  MoveL 7324 to (229.28, 36.09, 106.87) mm, rotated rx -180 ry 0 rz -180 deg; joints [-156.206, -68.965, -50.791, 41.618, 37.406, -35.211]
  MoveL 7325 to (229.28, 36.09, 106.87) mm, rotated rx -180 ry 0 rz -180 deg; joints [-156.206, -68.965, -50.791, 41.618, 37.406, -35.211]
  Call Extruder(199.41394)
  MoveL 7326 to (229.48, 36.14, 106.87) mm, rotated rx -180 ry 0 rz 180 deg; joints [-156.21, -68.992, -50.735, 41.638, 37.382, -35.238]
  MoveL 7327 to (229.48, 36.14, 106.87) mm, rotated rx -180 ry 0 rz 180 deg; joints [-156.21, -68.992, -50.735, 41.638, 37.382, -35.238]
  Call Extruder(199.52925)
  MoveL 7328 to (229.69, 36.18, 106.87) mm, rotated rx 180 ry 0 rz -180 deg; joints [-156.214, -69.019, -50.679, 41.658, 37.357, -35.266]
  MoveL 7329 to (229.69, 36.18, 106.87) mm, rotated rx 180 ry 0 rz -180 deg; joints [-156.214, -69.019, -50.679, 41.658, 37.357, -35.266]
  Call Extruder(199.65431)
  MoveL 7330 to (229.9, 36.25, 106.87) mm, rotated rx 180 ry 0 rz 180 deg; joints [-156.217, -69.048, -50.617, 41.682, 37.331, -35.299]
  MoveL 7331 to (229.9, 36.25, 106.87) mm, rotated rx 180 ry 0 rz 180 deg; joints [-156.217, -69.048, -50.617, 41.682, 37.331, -35.299]
  Call Extruder(199.77989)
  MoveL 7332 to (230.12, 36.31, 106.87) mm, rotated rx -180 ry 0 rz 180 deg; joints [-156.22, -69.077, -50.556, 41.707, 37.305, -35.331]
  MoveL 7333 to (230.12, 36.31, 106.87) mm, rotated rx -180 ry 0 rz 180 deg; joints [-156.22, -69.077, -50.556, 41.707, 37.305, -35.331]
  Call Extruder(199.90597)
  MoveL 7334 to (230.34, 36.37, 106.87) mm, rotated rx 180 ry 0 rz 180 deg; joints [-156.223, -69.106, -50.494, 41.731, 37.279, -35.364]
  MoveL 7335 to (230.34, 36.37, 106.87) mm, rotated rx 180 ry 0 rz 180 deg; joints [-156.223, -69.106, -50.494, 41.731, 37.279, -35.364]
  Call Extruder(200.01064)
  MoveL 7336 to (230.52, 36.43, 106.87) mm, rotated rx 180 ry 0 rz -180 deg; joints [-156.225, -69.131, -50.443, 41.752, 37.258, -35.391]
  MoveL 7337 to (230.52, 36.43, 106.87) mm, rotated rx 180 ry 0 rz -180 deg; joints [-156.225, -69.131, -50.443, 41.752, 37.258, -35.391]
  Call Extruder(200.11570)
  MoveL 7338 to (230.69, 36.49, 106.87) mm, rotated rx 180 ry 0 rz -180 deg; joints [-156.227, -69.155, -50.392, 41.773, 37.237, -35.419]
  MoveL 7339 to (230.69, 36.49, 106.87) mm, rotated rx 180 ry 0 rz -180 deg; joints [-156.227, -69.155, -50.392, 41.773, 37.237, -35.419]
  Call Extruder(200.22759)
  MoveL 7340 to (230.88, 36.55, 106.87) mm, rotated rx 180 ry 0 rz 180 deg; joints [-156.229, -69.181, -50.337, 41.795, 37.214, -35.448]
  MoveL 7341 to (230.88, 36.55, 106.87) mm, rotated rx 180 ry 0 rz 180 deg; joints [-156.229, -69.181, -50.337, 41.795, 37.214, -35.448]
  Call Extruder(200.33994)
  MoveL 7342 to (231.07, 36.61, 106.87) mm, rotated rx -180 ry 0 rz 180 deg; joints [-156.231, -69.207, -50.283, 41.818, 37.192, -35.477]
  MoveL 7343 to (231.07, 36.61, 106.87) mm, rotated rx -180 ry 0 rz 180 deg; joints [-156.231, -69.207, -50.283, 41.818, 37.192, -35.477]
  Call Extruder(200.45272)
  MoveL 7344 to (231.26, 36.67, 106.87) mm, rotated rx -180 ry 0 rz 180 deg; joints [-156.233, -69.232, -50.228, 41.84, 37.17, -35.507]
  MoveL 7345 to (231.26, 36.67, 106.87) mm, rotated rx -180 ry 0 rz 180 deg; joints [-156.233, -69.232, -50.228, 41.84, 37.17, -35.507]
  Call Extruder(200.56596)
  MoveL 7346 to (231.45, 36.73, 106.87) mm, rotated rx 180 ry 0 rz 180 deg; joints [-156.235, -69.258, -50.174, 41.863, 37.147, -35.536]
  MoveL 7347 to (231.45, 36.73, 106.87) mm, rotated rx 180 ry 0 rz 180 deg; joints [-156.235, -69.258, -50.174, 41.863, 37.147, -35.536]
  Call Extruder(200.67963)
  MoveL 7348 to (231.64, 36.79, 106.87) mm, rotated rx 180 ry 0 rz 180 deg; joints [-156.237, -69.284, -50.119, 41.885, 37.125, -35.566]
  MoveL 7349 to (231.64, 36.79, 106.87) mm, rotated rx 180 ry 0 rz 180 deg; joints [-156.237, -69.284, -50.119, 41.885, 37.125, -35.566]
  Call Extruder(200.86159)
  MoveL 7350 to (231.93, 36.91, 106.87) mm, rotated rx 180 ry 0 rz 180 deg; joints [-156.238, -69.326, -50.032, 41.925, 37.09, -35.616]
  MoveL 7351 to (231.93, 36.91, 106.87) mm, rotated rx 180 ry 0 rz 180 deg; joints [-156.238, -69.326, -50.032, 41.925, 37.09, -35.616]
  Call Extruder(201.04431)
  MoveL 7352 to (232.22, 37.03, 106.87) mm, rotated rx 180 ry 0 rz 180 deg; joints [-156.238, -69.367, -49.944, 41.965, 37.055, -35.666]
  MoveL 7353 to (232.22, 37.03, 106.87) mm, rotated rx 180 ry 0 rz 180 deg; joints [-156.238, -69.367, -49.944, 41.965, 37.055, -35.666]
  Call Extruder(201.21473)
  MoveL 7354 to (232.49, 37.15, 106.87) mm, rotated rx 180 ry 0 rz 180 deg; joints [-156.239, -69.406, -49.863, 42.002, 37.023, -35.713]
  MoveL 7355 to (232.49, 37.15, 106.87) mm, rotated rx 180 ry 0 rz 180 deg; joints [-156.239, -69.406, -49.863, 42.002, 37.023, -35.713]
  Call Extruder(201.37273)
  MoveL 7356 to (232.74, 37.26, 106.87) mm, rotated rx 180 ry 0 rz 180 deg; joints [-156.239, -69.442, -49.787, 42.037, 36.994, -35.757]
  MoveL 7357 to (232.74, 37.26, 106.87) mm, rotated rx 180 ry 0 rz 180 deg; joints [-156.239, -69.442, -49.787, 42.037, 36.994, -35.757]
  Call Extruder(201.53133)
  MoveL 7358 to (232.99, 37.36, 106.87) mm, rotated rx -180 ry 0 rz -180 deg; joints [-156.239, -69.478, -49.711, 42.072, 36.964, -35.801]
  MoveL 7359 to (232.99, 37.36, 106.87) mm, rotated rx -180 ry 0 rz -180 deg; joints [-156.239, -69.478, -49.711, 42.072, 36.964, -35.801]
  Call Extruder(201.73750)
  MoveL 7360 to (233.29, 37.54, 106.87) mm, rotated rx 180 ry 0 rz 180 deg; joints [-156.236, -69.524, -49.614, 42.122, 36.928, -35.862]
  MoveL 7361 to (233.29, 37.54, 106.87) mm, rotated rx 180 ry 0 rz 180 deg; joints [-156.236, -69.524, -49.614, 42.122, 36.928, -35.862]
  Call Extruder(201.94444)
  MoveL 7362 to (233.6, 37.71, 106.87) mm, rotated rx -180 ry 0 rz 180 deg; joints [-156.232, -69.57, -49.517, 42.173, 36.893, -35.923]
  MoveL 7363 to (233.6, 37.71, 106.87) mm, rotated rx -180 ry 0 rz 180 deg; joints [-156.232, -69.57, -49.517, 42.173, 36.893, -35.923]
  Call Extruder(202.15217)
  MoveL 7364 to (233.9, 37.89, 106.87) mm, rotated rx -180 ry 0 rz -180 deg; joints [-156.228, -69.617, -49.419, 42.224, 36.857, -35.984]
  MoveL 7365 to (233.9, 37.89, 106.87) mm, rotated rx -180 ry 0 rz -180 deg; joints [-156.228, -69.617, -49.419, 42.224, 36.857, -35.984]
  Call Extruder(202.36067)
  MoveL 7366 to (234.21, 38.06, 106.87) mm, rotated rx 180 ry 0 rz 180 deg; joints [-156.224, -69.663, -49.322, 42.275, 36.821, -36.046]
  MoveL 7367 to (234.21, 38.06, 106.87) mm, rotated rx 180 ry 0 rz 180 deg; joints [-156.224, -69.663, -49.322, 42.275, 36.821, -36.046]
  Call Extruder(202.54021)
  MoveL 7368 to (234.45, 38.24, 106.87) mm, rotated rx -180 ry 0 rz 180 deg; joints [-156.218, -69.703, -49.239, 42.322, 36.793, -36.101]
  MoveL 7369 to (234.45, 38.24, 106.87) mm, rotated rx -180 ry 0 rz 180 deg; joints [-156.218, -69.703, -49.239, 42.322, 36.793, -36.101]
  Call Extruder(202.87363)
  MoveL 7370 to (234.9, 38.57, 106.87) mm, rotated rx 180 ry 0 rz -180 deg; joints [-156.206, -69.776, -49.086, 42.411, 36.741, -36.204]
  MoveL 7371 to (234.9, 38.57, 106.87) mm, rotated rx 180 ry 0 rz -180 deg; joints [-156.206, -69.776, -49.086, 42.411, 36.741, -36.204]
  Call Extruder(203.20823)
  MoveL 7372 to (235.35, 38.9, 106.87) mm, rotated rx -180 ry 0 rz 180 deg; joints [-156.195, -69.849, -48.932, 42.499, 36.688, -36.308]
  Call Extruder(204.03618)
  MoveL 7373 to (236.39, 39.81, 106.87) mm, rotated rx 180 ry 0 rz 180 deg; joints [-156.154, -70.026, -48.56, 42.732, 36.569, -36.573]
  Call Extruder(204.86412)
  MoveL 7374 to (237.3, 40.85, 106.87) mm, rotated rx 180 ry 0 rz 180 deg; joints [-156.097, -70.196, -48.204, 42.98, 36.467, -36.848]
  Call Extruder(205.03142)
  MoveL 7375 to (237.47, 41.07, 106.87) mm, rotated rx 180 ry 0 rz 180 deg; joints [-156.083, -70.229, -48.135, 43.032, 36.449, -36.904]
  MoveL 7376 to (237.47, 41.07, 106.87) mm, rotated rx 180 ry 0 rz 180 deg; joints [-156.083, -70.229, -48.135, 43.032, 36.449, -36.904]
  Call Extruder(205.36483)
  MoveL 7377 to (237.8, 41.52, 106.87) mm, rotated rx 180 ry 0 rz 180 deg; joints [-156.055, -70.295, -47.997, 43.135, 36.412, -37.017]
  MoveL 7378 to (237.8, 41.52, 106.87) mm, rotated rx 180 ry 0 rz 180 deg; joints [-156.055, -70.295, -47.997, 43.135, 36.412, -37.017]
  Call Extruder(205.69706)
  MoveL 7379 to (238.12, 41.98, 106.87) mm, rotated rx 180 ry 0 rz -180 deg; joints [-156.028, -70.361, -47.858, 43.239, 36.376, -37.13]
  MoveL 7380 to (238.12, 41.98, 106.87) mm, rotated rx 180 ry 0 rz -180 deg; joints [-156.028, -70.361, -47.858, 43.239, 36.376, -37.13]
  Call Extruder(205.81476)
  MoveL 7381 to (238.22, 42.15, 106.87) mm, rotated rx -180 ry 0 rz -180 deg; joints [-156.016, -70.383, -47.813, 43.277, 36.366, -37.17]
  MoveL 7382 to (238.22, 42.15, 106.87) mm, rotated rx -180 ry 0 rz -180 deg; joints [-156.016, -70.383, -47.813, 43.277, 36.366, -37.17]
  Call Extruder(206.02249)
  MoveL 7383 to (238.4, 42.45, 106.87) mm, rotated rx 180 ry 0 rz 180 deg; joints [-155.996, -70.422, -47.731, 43.344, 36.347, -37.241]
  MoveL 7384 to (238.4, 42.45, 106.87) mm, rotated rx 180 ry 0 rz 180 deg; joints [-155.996, -70.422, -47.731, 43.344, 36.347, -37.241]
  Call Extruder(206.22943)
  MoveL 7385 to (238.57, 42.75, 106.87) mm, rotated rx -180 ry 0 rz -180 deg; joints [-155.976, -70.461, -47.65, 43.411, 36.328, -37.313]
  MoveL 7386 to (238.57, 42.75, 106.87) mm, rotated rx -180 ry 0 rz -180 deg; joints [-155.976, -70.461, -47.65, 43.411, 36.328, -37.313]
  Call Extruder(206.43560)
  MoveL 7387 to (238.75, 43.06, 106.87) mm, rotated rx 180 ry 0 rz 180 deg; joints [-155.956, -70.5, -47.568, 43.478, 36.31, -37.384]
  MoveL 7388 to (238.75, 43.06, 106.87) mm, rotated rx 180 ry 0 rz 180 deg; joints [-155.956, -70.5, -47.568, 43.478, 36.31, -37.384]
  Call Extruder(206.61728)
  MoveL 7389 to (238.89, 43.33, 106.87) mm, rotated rx 180 ry 0 rz 180 deg; joints [-155.937, -70.533, -47.498, 43.538, 36.295, -37.447]
  MoveL 7390 to (238.89, 43.33, 106.87) mm, rotated rx 180 ry 0 rz 180 deg; joints [-155.937, -70.533, -47.498, 43.538, 36.295, -37.447]
  Call Extruder(206.77529)
  MoveL 7391 to (239, 43.58, 106.87) mm, rotated rx -180 ry 0 rz -180 deg; joints [-155.919, -70.56, -47.441, 43.59, 36.284, -37.501]
  MoveL 7392 to (239, 43.58, 106.87) mm, rotated rx -180 ry 0 rz -180 deg; joints [-155.919, -70.56, -47.441, 43.59, 36.284, -37.501]
  Call Extruder(206.93270)
  MoveL 7393 to (239.1, 43.83, 106.87) mm, rotated rx 180 ry 0 rz -180 deg; joints [-155.901, -70.588, -47.383, 43.642, 36.273, -37.556]
  MoveL 7394 to (239.1, 43.83, 106.87) mm, rotated rx 180 ry 0 rz -180 deg; joints [-155.901, -70.588, -47.383, 43.642, 36.273, -37.556]
  Call Extruder(207.11542)
  MoveL 7395 to (239.23, 44.12, 106.87) mm, rotated rx 180 ry 0 rz 180 deg; joints [-155.879, -70.619, -47.317, 43.703, 36.261, -37.619]
  MoveL 7396 to (239.23, 44.12, 106.87) mm, rotated rx 180 ry 0 rz 180 deg; joints [-155.879, -70.619, -47.317, 43.703, 36.261, -37.619]
  Call Extruder(207.29737)
  MoveL 7397 to (239.35, 44.42, 106.87) mm, rotated rx 180 ry 0 rz -180 deg; joints [-155.858, -70.651, -47.251, 43.764, 36.249, -37.682]
  MoveL 7398 to (239.35, 44.42, 106.87) mm, rotated rx 180 ry 0 rz -180 deg; joints [-155.858, -70.651, -47.251, 43.764, 36.249, -37.682]
  Call Extruder(207.44470)
  MoveL 7399 to (239.44, 44.66, 106.87) mm, rotated rx -180 ry 0 rz -180 deg; joints [-155.84, -70.676, -47.199, 43.814, 36.241, -37.734]
  MoveL 7400 to (239.44, 44.66, 106.87) mm, rotated rx -180 ry 0 rz -180 deg; joints [-155.84, -70.676, -47.199, 43.814, 36.241, -37.734]
  Call Extruder(207.55794)
  MoveL 7401 to (239.5, 44.85, 106.87) mm, rotated rx -180 ry 0 rz 180 deg; joints [-155.826, -70.695, -47.16, 43.852, 36.235, -37.773]
  MoveL 7402 to (239.5, 44.85, 106.87) mm, rotated rx -180 ry 0 rz 180 deg; joints [-155.826, -70.695, -47.16, 43.852, 36.235, -37.773]
  Call Extruder(207.67073)
  MoveL 7403 to (239.56, 45.03, 106.87) mm, rotated rx -180 ry 0 rz 180 deg; joints [-155.811, -70.713, -47.121, 43.89, 36.229, -37.812]
  MoveL 7404 to (239.56, 45.03, 106.87) mm, rotated rx -180 ry 0 rz 180 deg; joints [-155.811, -70.713, -47.121, 43.89, 36.229, -37.812]
  Call Extruder(207.78308)
  MoveL 7405 to (239.62, 45.22, 106.87) mm, rotated rx 180 ry 0 rz -180 deg; joints [-155.797, -70.732, -47.083, 43.929, 36.224, -37.851]
  MoveL 7406 to (239.62, 45.22, 106.87) mm, rotated rx 180 ry 0 rz -180 deg; joints [-155.797, -70.732, -47.083, 43.929, 36.224, -37.851]
  Call Extruder(207.89498)
  MoveL 7407 to (239.68, 45.41, 106.87) mm, rotated rx -180 ry 0 rz 180 deg; joints [-155.783, -70.75, -47.044, 43.967, 36.218, -37.89]
  MoveL 7408 to (239.68, 45.41, 106.87) mm, rotated rx -180 ry 0 rz 180 deg; joints [-155.783, -70.75, -47.044, 43.967, 36.218, -37.89]
  Call Extruder(208.01638)
  MoveL 7409 to (239.75, 45.62, 106.87) mm, rotated rx 180 ry 0 rz 180 deg; joints [-155.767, -70.77, -47.003, 44.009, 36.212, -37.932]
  MoveL 7410 to (239.75, 45.62, 106.87) mm, rotated rx 180 ry 0 rz 180 deg; joints [-155.767, -70.77, -47.003, 44.009, 36.212, -37.932]
  Call Extruder(208.14717)
  MoveL 7411 to (239.81, 45.84, 106.87) mm, rotated rx 180 ry 0 rz 180 deg; joints [-155.75, -70.791, -46.958, 44.054, 36.206, -37.978]
  MoveL 7412 to (239.81, 45.84, 106.87) mm, rotated rx 180 ry 0 rz 180 deg; joints [-155.75, -70.791, -46.958, 44.054, 36.206, -37.978]
  Call Extruder(208.27740)
  MoveL 7413 to (239.88, 46.06, 106.87) mm, rotated rx 180 ry 0 rz 180 deg; joints [-155.733, -70.813, -46.914, 44.099, 36.2, -38.024]
  MoveL 7414 to (239.88, 46.06, 106.87) mm, rotated rx 180 ry 0 rz 180 deg; joints [-155.733, -70.813, -46.914, 44.099, 36.2, -38.024]
  Call Extruder(208.40706)
  MoveL 7415 to (239.95, 46.29, 106.87) mm, rotated rx -180 ry 0 rz 180 deg; joints [-155.715, -70.834, -46.869, 44.144, 36.194, -38.07]
  MoveL 7416 to (239.95, 46.29, 106.87) mm, rotated rx -180 ry 0 rz 180 deg; joints [-155.715, -70.834, -46.869, 44.144, 36.194, -38.07]
  Call Extruder(208.53615)
  MoveL 7417 to (240.02, 46.51, 106.87) mm, rotated rx 180 ry 0 rz 180 deg; joints [-155.698, -70.855, -46.824, 44.189, 36.188, -38.116]
  MoveL 7418 to (240.02, 46.51, 106.87) mm, rotated rx 180 ry 0 rz 180 deg; joints [-155.698, -70.855, -46.824, 44.189, 36.188, -38.116]
  Call Extruder(208.65121)
  MoveL 7419 to (240.06, 46.72, 106.87) mm, rotated rx -180 ry 0 rz -180 deg; joints [-155.682, -70.873, -46.788, 44.229, 36.184, -38.156]
  MoveL 7420 to (240.06, 46.72, 106.87) mm, rotated rx -180 ry 0 rz -180 deg; joints [-155.682, -70.873, -46.788, 44.229, 36.184, -38.156]
  Call Extruder(208.76581)
  MoveL 7421 to (240.11, 46.92, 106.87) mm, rotated rx 180 ry 0 rz -180 deg; joints [-155.665, -70.89, -46.751, 44.269, 36.181, -38.196]
  MoveL 7422 to (240.11, 46.92, 106.87) mm, rotated rx 180 ry 0 rz -180 deg; joints [-155.665, -70.89, -46.751, 44.269, 36.181, -38.196]
  Call Extruder(208.87996)
  MoveL 7423 to (240.15, 47.12, 106.87) mm, rotated rx 180 ry 0 rz 180 deg; joints [-155.649, -70.908, -46.715, 44.308, 36.177, -38.236]
  MoveL 7424 to (240.15, 47.12, 106.87) mm, rotated rx 180 ry 0 rz 180 deg; joints [-155.649, -70.908, -46.715, 44.308, 36.177, -38.236]
  Call Extruder(208.99365)
  MoveL 7425 to (240.2, 47.33, 106.87) mm, rotated rx 180 ry 0 rz 180 deg; joints [-155.633, -70.925, -46.679, 44.348, 36.174, -38.276]
  MoveL 7426 to (240.2, 47.33, 106.87) mm, rotated rx 180 ry 0 rz 180 deg; joints [-155.633, -70.925, -46.679, 44.348, 36.174, -38.276]
  Call Extruder(209.11906)
  MoveL 7427 to (240.24, 47.55, 106.87) mm, rotated rx 180 ry 0 rz 180 deg; joints [-155.614, -70.944, -46.639, 44.392, 36.17, -38.32]
  MoveL 7428 to (240.24, 47.55, 106.87) mm, rotated rx 180 ry 0 rz 180 deg; joints [-155.614, -70.944, -46.639, 44.392, 36.17, -38.32]
  Call Extruder(209.25604)
  MoveL 7429 to (240.29, 47.8, 106.87) mm, rotated rx -180 ry 0 rz 180 deg; joints [-155.594, -70.965, -46.596, 44.441, 36.167, -38.369]
  MoveL 7430 to (240.29, 47.8, 106.87) mm, rotated rx -180 ry 0 rz 180 deg; joints [-155.594, -70.965, -46.596, 44.441, 36.167, -38.369]
  Call Extruder(209.39241)
  MoveL 7431 to (240.34, 48.05, 106.87) mm, rotated rx 180 ry 0 rz 180 deg; joints [-155.574, -70.986, -46.553, 44.489, 36.163, -38.417]
  MoveL 7432 to (240.34, 48.05, 106.87) mm, rotated rx 180 ry 0 rz 180 deg; joints [-155.574, -70.986, -46.553, 44.489, 36.163, -38.417]
  Call Extruder(209.52817)
  MoveL 7433 to (240.39, 48.3, 106.87) mm, rotated rx 180 ry 0 rz 180 deg; joints [-155.554, -71.006, -46.509, 44.538, 36.159, -38.465]
  MoveL 7434 to (240.39, 48.3, 106.87) mm, rotated rx 180 ry 0 rz 180 deg; joints [-155.554, -71.006, -46.509, 44.538, 36.159, -38.465]
  Call Extruder(209.66331)
  MoveL 7435 to (240.44, 48.55, 106.87) mm, rotated rx -180 ry 0 rz 180 deg; joints [-155.534, -71.027, -46.466, 44.586, 36.156, -38.514]
  MoveL 7436 to (240.44, 48.55, 106.87) mm, rotated rx -180 ry 0 rz 180 deg; joints [-155.534, -71.027, -46.466, 44.586, 36.156, -38.514]
  Call Extruder(209.79785)
  MoveL 7437 to (240.49, 48.8, 106.87) mm, rotated rx -180 ry 0 rz -180 deg; joints [-155.514, -71.048, -46.422, 44.634, 36.152, -38.562]
  MoveL 7438 to (240.49, 48.8, 106.87) mm, rotated rx -180 ry 0 rz -180 deg; joints [-155.514, -71.048, -46.422, 44.634, 36.152, -38.562]
  Call Extruder(209.93178)
  MoveL 7439 to (240.54, 49.05, 106.87) mm, rotated rx 180 ry 0 rz 180 deg; joints [-155.494, -71.069, -46.379, 44.683, 36.149, -38.61]
  MoveL 7440 to (240.54, 49.05, 106.87) mm, rotated rx 180 ry 0 rz 180 deg; joints [-155.494, -71.069, -46.379, 44.683, 36.149, -38.61]
  Call Extruder(210.07964)
  MoveL 7441 to (240.59, 49.33, 106.87) mm, rotated rx 180 ry 0 rz 180 deg; joints [-155.471, -71.091, -46.332, 44.736, 36.146, -38.664]
  MoveL 7442 to (240.59, 49.33, 106.87) mm, rotated rx 180 ry 0 rz 180 deg; joints [-155.471, -71.091, -46.332, 44.736, 36.146, -38.664]
  Call Extruder(210.24139)
  MoveL 7443 to (240.64, 49.63, 106.87) mm, rotated rx 180 ry 0 rz -180 deg; joints [-155.446, -71.115, -46.282, 44.794, 36.143, -38.722]
  MoveL 7444 to (240.64, 49.63, 106.87) mm, rotated rx 180 ry 0 rz -180 deg; joints [-155.446, -71.115, -46.282, 44.794, 36.143, -38.722]
  Call Extruder(210.40241)
  MoveL 7445 to (240.69, 49.94, 106.87) mm, rotated rx 180 ry 0 rz 180 deg; joints [-155.421, -71.139, -46.232, 44.853, 36.14, -38.78]
  MoveL 7446 to (240.69, 49.94, 106.87) mm, rotated rx 180 ry 0 rz 180 deg; joints [-155.421, -71.139, -46.232, 44.853, 36.14, -38.78]
  Call Extruder(210.56270)
  MoveL 7447 to (240.74, 50.24, 106.87) mm, rotated rx 180 ry 0 rz 180 deg; joints [-155.396, -71.164, -46.181, 44.911, 36.137, -38.838]
  MoveL 7448 to (240.74, 50.24, 106.87) mm, rotated rx 180 ry 0 rz 180 deg; joints [-155.396, -71.164, -46.181, 44.911, 36.137, -38.838]
  Call Extruder(210.72226)
  MoveL 7449 to (240.78, 50.55, 106.87) mm, rotated rx 180 ry 0 rz 180 deg; joints [-155.371, -71.188, -46.131, 44.97, 36.134, -38.896]
  MoveL 7450 to (240.78, 50.55, 106.87) mm, rotated rx 180 ry 0 rz 180 deg; joints [-155.371, -71.188, -46.131, 44.97, 36.134, -38.896]
  Call Extruder(210.88109)
  MoveL 7451 to (240.83, 50.86, 106.87) mm, rotated rx 180 ry 0 rz 180 deg; joints [-155.346, -71.212, -46.08, 45.028, 36.131, -38.954]
  MoveL 7452 to (240.83, 50.86, 106.87) mm, rotated rx 180 ry 0 rz 180 deg; joints [-155.346, -71.212, -46.08, 45.028, 36.131, -38.954]
  Call Extruder(211.05976)
  MoveL 7453 to (240.88, 51.2, 106.87) mm, rotated rx -180 ry 0 rz -180 deg; joints [-155.317, -71.238, -46.025, 45.094, 36.129, -39.019]
  MoveL 7454 to (240.88, 51.2, 106.87) mm, rotated rx -180 ry 0 rz -180 deg; joints [-155.317, -71.238, -46.025, 45.094, 36.129, -39.019]
  Call Extruder(211.25821)
  MoveL 7455 to (240.93, 51.59, 106.87) mm, rotated rx 180 ry 0 rz -180 deg; joints [-155.285, -71.267, -45.965, 45.167, 36.127, -39.091]
  MoveL 7456 to (240.93, 51.59, 106.87) mm, rotated rx 180 ry 0 rz -180 deg; joints [-155.285, -71.267, -45.965, 45.167, 36.127, -39.091]
  Call Extruder(211.45578)
  MoveL 7457 to (240.97, 51.98, 106.87) mm, rotated rx -180 ry 0 rz 180 deg; joints [-155.252, -71.296, -45.905, 45.24, 36.126, -39.163]
  MoveL 7458 to (240.97, 51.98, 106.87) mm, rotated rx -180 ry 0 rz 180 deg; joints [-155.252, -71.296, -45.905, 45.24, 36.126, -39.163]
  Call Extruder(211.65249)
  MoveL 7459 to (241.02, 52.36, 106.87) mm, rotated rx -180 ry 0 rz 180 deg; joints [-155.22, -71.325, -45.845, 45.313, 36.124, -39.235]
  MoveL 7460 to (241.02, 52.36, 106.87) mm, rotated rx -180 ry 0 rz 180 deg; joints [-155.22, -71.325, -45.845, 45.313, 36.124, -39.235]
  Call Extruder(211.84833)
  MoveL 7461 to (241.06, 52.75, 106.87) mm, rotated rx 180 ry 0 rz 180 deg; joints [-155.188, -71.354, -45.785, 45.386, 36.123, -39.307]
  MoveL 7462 to (241.06, 52.75, 106.87) mm, rotated rx 180 ry 0 rz 180 deg; joints [-155.188, -71.354, -45.785, 45.386, 36.123, -39.307]
  Call Extruder(212.14376)
  MoveL 7463 to (241.11, 53.34, 106.87) mm, rotated rx 180 ry 0 rz 180 deg; joints [-155.138, -71.395, -45.699, 45.495, 36.123, -39.414]
  MoveL 7464 to (241.11, 53.34, 106.87) mm, rotated rx 180 ry 0 rz 180 deg; joints [-155.138, -71.395, -45.699, 45.495, 36.123, -39.414]
  Call Extruder(212.43787)
  MoveL 7465 to (241.16, 53.93, 106.87) mm, rotated rx 180 ry 0 rz 180 deg; joints [-155.088, -71.436, -45.613, 45.604, 36.124, -39.521]
  MoveL 7466 to (241.16, 53.93, 106.87) mm, rotated rx 180 ry 0 rz 180 deg; joints [-155.088, -71.436, -45.613, 45.604, 36.124, -39.521]
  Call Extruder(212.73064)
  MoveL 7467 to (241.2, 54.52, 106.87) mm, rotated rx -180 ry 0 rz -180 deg; joints [-155.038, -71.478, -45.526, 45.713, 36.124, -39.629]
  MoveL 7468 to (241.2, 54.52, 106.87) mm, rotated rx -180 ry 0 rz -180 deg; joints [-155.038, -71.478, -45.526, 45.713, 36.124, -39.629]
  Call Extruder(213.30409)
  MoveL 7469 to (241.25, 55.68, 106.87) mm, rotated rx -180 ry 0 rz -180 deg; joints [-154.938, -71.554, -45.368, 45.925, 36.131, -39.834]
  MoveL 7470 to (241.25, 55.68, 106.87) mm, rotated rx -180 ry 0 rz -180 deg; joints [-154.938, -71.554, -45.368, 45.925, 36.131, -39.834]
  Call Extruder(214.01793)
  MoveL 7471 to (241.29, 57.14, 106.87) mm, rotated rx 180 ry 0 rz 180 deg; joints [-154.812, -71.648, -45.173, 46.188, 36.141, -40.09]
  Call Extruder(256.08281)
  MoveL 7472 to (241.29, 142.86, 106.87) mm, rotated rx 180 ry 0 rz 180 deg; joints [-147.778, -78.434, -31.275, 61.849, 37.21, -56.104]
  Call Extruder(256.51124)
  MoveL 7473 to (241.27, 143.73, 106.87) mm, rotated rx 180 ry 0 rz 180 deg; joints [-147.711, -78.521, -31.1, 62.014, 37.224, -56.283]
  MoveL 7474 to (241.27, 143.73, 106.87) mm, rotated rx 180 ry 0 rz 180 deg; joints [-147.711, -78.521, -31.1, 62.014, 37.224, -56.283]
  Call Extruder(257.08469)
  MoveL 7475 to (241.22, 144.9, 106.87) mm, rotated rx 180 ry 0 rz 180 deg; joints [-147.62, -78.634, -30.873, 62.231, 37.246, -56.517]
  MoveL 7476 to (241.22, 144.9, 106.87) mm, rotated rx 180 ry 0 rz 180 deg; joints [-147.62, -78.634, -30.873, 62.231, 37.246, -56.517]
  Call Extruder(257.51903)
  MoveL 7477 to (241.18, 145.77, 106.87) mm, rotated rx -180 ry 0 rz 180 deg; joints [-147.551, -78.717, -30.704, 62.393, 37.264, -56.691]
  MoveL 7478 to (241.18, 145.77, 106.87) mm, rotated rx -180 ry 0 rz 180 deg; joints [-147.551, -78.717, -30.704, 62.393, 37.264, -56.691]
  Call Extruder(257.81314)
  MoveL 7479 to (241.13, 146.36, 106.87) mm, rotated rx 180 ry 0 rz -180 deg; joints [-147.504, -78.771, -30.595, 62.499, 37.278, -56.805]
  MoveL 7480 to (241.13, 146.36, 106.87) mm, rotated rx 180 ry 0 rz -180 deg; joints [-147.504, -78.771, -30.595, 62.499, 37.278, -56.805]
  Call Extruder(258.10858)
  MoveL 7481 to (241.09, 146.95, 106.87) mm, rotated rx 180 ry 0 rz 180 deg; joints [-147.457, -78.825, -30.486, 62.606, 37.292, -56.92]
  MoveL 7482 to (241.09, 146.95, 106.87) mm, rotated rx 180 ry 0 rz 180 deg; joints [-147.457, -78.825, -30.486, 62.606, 37.292, -56.92]
  Call Extruder(258.35483)
  MoveL 7483 to (241.04, 147.44, 106.87) mm, rotated rx 180 ry 0 rz 180 deg; joints [-147.417, -78.869, -30.397, 62.693, 37.305, -57.013]
  MoveL 7484 to (241.04, 147.44, 106.87) mm, rotated rx 180 ry 0 rz 180 deg; joints [-147.417, -78.869, -30.397, 62.693, 37.305, -57.013]
  Call Extruder(258.55154)
  MoveL 7485 to (240.99, 147.83, 106.87) mm, rotated rx 180 ry 0 rz -180 deg; joints [-147.386, -78.903, -30.33, 62.761, 37.316, -57.086]
  MoveL 7486 to (240.99, 147.83, 106.87) mm, rotated rx 180 ry 0 rz -180 deg; joints [-147.386, -78.903, -30.33, 62.761, 37.316, -57.086]
  Call Extruder(258.74911)
  MoveL 7487 to (240.95, 148.22, 106.87) mm, rotated rx 180 ry 0 rz 180 deg; joints [-147.354, -78.936, -30.263, 62.829, 37.327, -57.158]
  MoveL 7488 to (240.95, 148.22, 106.87) mm, rotated rx 180 ry 0 rz 180 deg; joints [-147.354, -78.936, -30.263, 62.829, 37.327, -57.158]
  Call Extruder(258.94755)
  MoveL 7489 to (240.9, 148.6, 106.87) mm, rotated rx 180 ry 0 rz -180 deg; joints [-147.322, -78.969, -30.195, 62.897, 37.338, -57.23]
  MoveL 7490 to (240.9, 148.6, 106.87) mm, rotated rx 180 ry 0 rz -180 deg; joints [-147.322, -78.969, -30.195, 62.897, 37.338, -57.23]
  Call Extruder(259.14686)
  MoveL 7491 to (240.86, 148.99, 106.87) mm, rotated rx 180 ry 0 rz 180 deg; joints [-147.291, -79.003, -30.128, 62.965, 37.349, -57.303]
  MoveL 7492 to (240.86, 148.99, 106.87) mm, rotated rx 180 ry 0 rz 180 deg; joints [-147.291, -79.003, -30.128, 62.965, 37.349, -57.303]
  Call Extruder(259.30569)
  MoveL 7493 to (240.81, 149.3, 106.87) mm, rotated rx 180 ry 0 rz 180 deg; joints [-147.265, -79.028, -30.078, 63.017, 37.359, -57.357]
  MoveL 7494 to (240.81, 149.3, 106.87) mm, rotated rx 180 ry 0 rz 180 deg; joints [-147.265, -79.028, -30.078, 63.017, 37.359, -57.357]
  Call Extruder(259.46525)
  MoveL 7495 to (240.76, 149.6, 106.87) mm, rotated rx -180 ry 0 rz 180 deg; joints [-147.24, -79.052, -30.028, 63.068, 37.369, -57.412]
  MoveL 7496 to (240.76, 149.6, 106.87) mm, rotated rx -180 ry 0 rz 180 deg; joints [-147.24, -79.052, -30.028, 63.068, 37.369, -57.412]
  Call Extruder(259.62554)
  MoveL 7497 to (240.71, 149.91, 106.87) mm, rotated rx 180 ry 0 rz -180 deg; joints [-147.214, -79.077, -29.979, 63.12, 37.379, -57.467]
  MoveL 7498 to (240.71, 149.91, 106.87) mm, rotated rx 180 ry 0 rz -180 deg; joints [-147.214, -79.077, -29.979, 63.12, 37.379, -57.467]
  Call Extruder(259.78655)
  MoveL 7499 to (240.66, 150.21, 106.87) mm, rotated rx 180 ry 0 rz 180 deg; joints [-147.189, -79.102, -29.929, 63.172, 37.39, -57.521]
  MoveL 7500 to (240.66, 150.21, 106.87) mm, rotated rx 180 ry 0 rz 180 deg; joints [-147.189, -79.102, -29.929, 63.172, 37.39, -57.521]
  Call Extruder(259.94830)
  MoveL 7501 to (240.61, 150.52, 106.87) mm, rotated rx -180 ry 0 rz -180 deg; joints [-147.163, -79.126, -29.879, 63.224, 37.4, -57.576]
  MoveL 7502 to (240.61, 150.52, 106.87) mm, rotated rx -180 ry 0 rz -180 deg; joints [-147.163, -79.126, -29.879, 63.224, 37.4, -57.576]
  Call Extruder(260.11077)
  MoveL 7503 to (240.56, 150.83, 106.87) mm, rotated rx -180 ry 0 rz -180 deg; joints [-147.138, -79.151, -29.829, 63.276, 37.41, -57.631]
  MoveL 7504 to (240.56, 150.83, 106.87) mm, rotated rx -180 ry 0 rz -180 deg; joints [-147.138, -79.151, -29.829, 63.276, 37.41, -57.631]
  Call Extruder(260.24469)
  MoveL 7505 to (240.52, 151.07, 106.87) mm, rotated rx 180 ry 0 rz 180 deg; joints [-147.117, -79.17, -29.791, 63.317, 37.419, -57.674]
  MoveL 7506 to (240.52, 151.07, 106.87) mm, rotated rx 180 ry 0 rz 180 deg; joints [-147.117, -79.17, -29.791, 63.317, 37.419, -57.674]
  Call Extruder(260.37923)
  MoveL 7507 to (240.47, 151.32, 106.87) mm, rotated rx -180 ry 0 rz 180 deg; joints [-147.095, -79.188, -29.754, 63.357, 37.429, -57.716]
  MoveL 7508 to (240.47, 151.32, 106.87) mm, rotated rx -180 ry 0 rz 180 deg; joints [-147.095, -79.188, -29.754, 63.357, 37.429, -57.716]
  Call Extruder(260.51438)
  MoveL 7509 to (240.42, 151.57, 106.87) mm, rotated rx 180 ry 0 rz 180 deg; joints [-147.074, -79.207, -29.717, 63.398, 37.438, -57.759]
  MoveL 7510 to (240.42, 151.57, 106.87) mm, rotated rx 180 ry 0 rz 180 deg; joints [-147.074, -79.207, -29.717, 63.398, 37.438, -57.759]
  Call Extruder(260.65014)
  MoveL 7511 to (240.37, 151.82, 106.87) mm, rotated rx 180 ry 0 rz -180 deg; joints [-147.053, -79.226, -29.679, 63.439, 37.448, -57.802]
  MoveL 7512 to (240.37, 151.82, 106.87) mm, rotated rx 180 ry 0 rz -180 deg; joints [-147.053, -79.226, -29.679, 63.439, 37.448, -57.802]
  Call Extruder(260.78650)
  MoveL 7513 to (240.32, 152.07, 106.87) mm, rotated rx 180 ry 0 rz 180 deg; joints [-147.032, -79.244, -29.641, 63.479, 37.457, -57.844]
  MoveL 7514 to (240.32, 152.07, 106.87) mm, rotated rx 180 ry 0 rz 180 deg; joints [-147.032, -79.244, -29.641, 63.479, 37.457, -57.844]
  Call Extruder(260.92348)
  MoveL 7515 to (240.27, 152.32, 106.87) mm, rotated rx -180 ry 0 rz 180 deg; joints [-147.011, -79.263, -29.603, 63.52, 37.467, -57.887]
  MoveL 7516 to (240.27, 152.32, 106.87) mm, rotated rx -180 ry 0 rz 180 deg; joints [-147.011, -79.263, -29.603, 63.52, 37.467, -57.887]
  Call Extruder(261.06107)
  MoveL 7517 to (240.22, 152.57, 106.87) mm, rotated rx -180 ry 0 rz 180 deg; joints [-146.989, -79.282, -29.566, 63.561, 37.476, -57.929]
  MoveL 7518 to (240.22, 152.57, 106.87) mm, rotated rx -180 ry 0 rz 180 deg; joints [-146.989, -79.282, -29.566, 63.561, 37.476, -57.929]
  Call Extruder(261.17477)
  MoveL 7519 to (240.17, 152.77, 106.87) mm, rotated rx 180 ry 0 rz 180 deg; joints [-146.972, -79.297, -29.536, 63.594, 37.484, -57.964]
  MoveL 7520 to (240.17, 152.77, 106.87) mm, rotated rx 180 ry 0 rz 180 deg; joints [-146.972, -79.297, -29.536, 63.594, 37.484, -57.964]
  Call Extruder(261.28892)
  MoveL 7521 to (240.13, 152.98, 106.87) mm, rotated rx -180 ry 0 rz -180 deg; joints [-146.954, -79.312, -29.506, 63.626, 37.493, -57.998]
  MoveL 7522 to (240.13, 152.98, 106.87) mm, rotated rx -180 ry 0 rz -180 deg; joints [-146.954, -79.312, -29.506, 63.626, 37.493, -57.998]
  Call Extruder(261.40352)
  MoveL 7523 to (240.08, 153.18, 106.87) mm, rotated rx -180 ry 0 rz 180 deg; joints [-146.937, -79.326, -29.476, 63.659, 37.501, -58.032]
  MoveL 7524 to (240.08, 153.18, 106.87) mm, rotated rx -180 ry 0 rz 180 deg; joints [-146.937, -79.326, -29.476, 63.659, 37.501, -58.032]
  Call Extruder(261.51858)
  MoveL 7525 to (240.04, 153.39, 106.87) mm, rotated rx 180 ry 0 rz -180 deg; joints [-146.919, -79.341, -29.446, 63.692, 37.509, -58.066]
  MoveL 7526 to (240.04, 153.39, 106.87) mm, rotated rx 180 ry 0 rz -180 deg; joints [-146.919, -79.341, -29.446, 63.692, 37.509, -58.066]
  Call Extruder(261.64080)
  MoveL 7527 to (239.98, 153.6, 106.87) mm, rotated rx 180 ry 0 rz 180 deg; joints [-146.9, -79.355, -29.418, 63.725, 37.519, -58.1]
  MoveL 7528 to (239.98, 153.6, 106.87) mm, rotated rx 180 ry 0 rz 180 deg; joints [-146.9, -79.355, -29.418, 63.725, 37.519, -58.1]
  Call Extruder(261.77046)
  MoveL 7529 to (239.92, 153.82, 106.87) mm, rotated rx 180 ry 0 rz 180 deg; joints [-146.88, -79.369, -29.392, 63.758, 37.53, -58.134]
  MoveL 7530 to (239.92, 153.82, 106.87) mm, rotated rx 180 ry 0 rz 180 deg; joints [-146.88, -79.369, -29.392, 63.758, 37.53, -58.134]
  Call Extruder(261.90069)
  MoveL 7531 to (239.85, 154.05, 106.87) mm, rotated rx -180 ry 0 rz 180 deg; joints [-146.86, -79.382, -29.366, 63.791, 37.541, -58.167]
  MoveL 7532 to (239.85, 154.05, 106.87) mm, rotated rx -180 ry 0 rz 180 deg; joints [-146.86, -79.382, -29.366, 63.791, 37.541, -58.167]
  Call Extruder(262.03148)
  MoveL 7533 to (239.78, 154.27, 106.87) mm, rotated rx 180 ry 0 rz -180 deg; joints [-146.84, -79.395, -29.339, 63.824, 37.553, -58.201]
  MoveL 7534 to (239.78, 154.27, 106.87) mm, rotated rx 180 ry 0 rz -180 deg; joints [-146.84, -79.395, -29.339, 63.824, 37.553, -58.201]
  Call Extruder(262.16284)
  MoveL 7535 to (239.71, 154.49, 106.87) mm, rotated rx 180 ry 0 rz 180 deg; joints [-146.82, -79.408, -29.312, 63.857, 37.564, -58.234]
  MoveL 7536 to (239.71, 154.49, 106.87) mm, rotated rx 180 ry 0 rz 180 deg; joints [-146.82, -79.408, -29.312, 63.857, 37.564, -58.234]
  Call Extruder(262.27474)
  MoveL 7537 to (239.65, 154.68, 106.87) mm, rotated rx 180 ry 0 rz 180 deg; joints [-146.803, -79.419, -29.291, 63.884, 37.574, -58.261]
  MoveL 7538 to (239.65, 154.68, 106.87) mm, rotated rx 180 ry 0 rz 180 deg; joints [-146.803, -79.419, -29.291, 63.884, 37.574, -58.261]
  Call Extruder(262.38708)
  MoveL 7539 to (239.59, 154.87, 106.87) mm, rotated rx -180 ry 0 rz 180 deg; joints [-146.785, -79.429, -29.27, 63.911, 37.584, -58.289]
  MoveL 7540 to (239.59, 154.87, 106.87) mm, rotated rx -180 ry 0 rz 180 deg; joints [-146.785, -79.429, -29.27, 63.911, 37.584, -58.289]
  Call Extruder(262.49987)
  MoveL 7541 to (239.53, 155.06, 106.87) mm, rotated rx 180 ry 0 rz 180 deg; joints [-146.768, -79.439, -29.249, 63.938, 37.594, -58.316]
  MoveL 7542 to (239.53, 155.06, 106.87) mm, rotated rx 180 ry 0 rz 180 deg; joints [-146.768, -79.439, -29.249, 63.938, 37.594, -58.316]
  Call Extruder(262.61311)
  MoveL 7543 to (239.47, 155.25, 106.87) mm, rotated rx 180 ry 0 rz 180 deg; joints [-146.751, -79.45, -29.228, 63.966, 37.604, -58.343]
  MoveL 7544 to (239.47, 155.25, 106.87) mm, rotated rx 180 ry 0 rz 180 deg; joints [-146.751, -79.45, -29.228, 63.966, 37.604, -58.343]
  Call Extruder(262.72679)
  MoveL 7545 to (239.41, 155.44, 106.87) mm, rotated rx -180 ry 0 rz 180 deg; joints [-146.734, -79.461, -29.207, 63.993, 37.613, -58.371]
  MoveL 7546 to (239.41, 155.44, 106.87) mm, rotated rx -180 ry 0 rz 180 deg; joints [-146.734, -79.461, -29.207, 63.993, 37.613, -58.371]
  Call Extruder(262.90875)
  MoveL 7547 to (239.29, 155.73, 106.87) mm, rotated rx -180 ry 0 rz 180 deg; joints [-146.706, -79.472, -29.183, 64.031, 37.632, -58.407]
  MoveL 7548 to (239.29, 155.73, 106.87) mm, rotated rx -180 ry 0 rz 180 deg; joints [-146.706, -79.472, -29.183, 64.031, 37.632, -58.407]
  Call Extruder(263.09146)
  MoveL 7549 to (239.16, 156.02, 106.87) mm, rotated rx -180 ry 0 rz 180 deg; joints [-146.678, -79.484, -29.159, 64.069, 37.65, -58.444]
  MoveL 7550 to (239.16, 156.02, 106.87) mm, rotated rx -180 ry 0 rz 180 deg; joints [-146.678, -79.484, -29.159, 64.069, 37.65, -58.444]
  Call Extruder(263.26189)
  MoveL 7551 to (239.05, 156.29, 106.87) mm, rotated rx 180 ry 0 rz -180 deg; joints [-146.652, -79.495, -29.137, 64.103, 37.668, -58.478]
  MoveL 7552 to (239.05, 156.29, 106.87) mm, rotated rx 180 ry 0 rz -180 deg; joints [-146.652, -79.495, -29.137, 64.103, 37.668, -58.478]
  Call Extruder(263.41990)
  MoveL 7553 to (238.94, 156.54, 106.87) mm, rotated rx 180 ry 0 rz 180 deg; joints [-146.628, -79.505, -29.118, 64.135, 37.684, -58.508]
  MoveL 7554 to (238.94, 156.54, 106.87) mm, rotated rx 180 ry 0 rz 180 deg; joints [-146.628, -79.505, -29.118, 64.135, 37.684, -58.508]
  Call Extruder(263.57851)
  MoveL 7555 to (238.84, 156.79, 106.87) mm, rotated rx 180 ry 0 rz 180 deg; joints [-146.604, -79.514, -29.098, 64.167, 37.7, -58.539]
  MoveL 7556 to (238.84, 156.79, 106.87) mm, rotated rx 180 ry 0 rz 180 deg; joints [-146.604, -79.514, -29.098, 64.167, 37.7, -58.539]
  Call Extruder(263.78468)
  MoveL 7557 to (238.66, 157.09, 106.87) mm, rotated rx -180 ry 0 rz 180 deg; joints [-146.573, -79.519, -29.09, 64.199, 37.725, -58.566]
  MoveL 7558 to (238.66, 157.09, 106.87) mm, rotated rx -180 ry 0 rz 180 deg; joints [-146.573, -79.519, -29.09, 64.199, 37.725, -58.566]
  Call Extruder(263.99163)
  MoveL 7559 to (238.49, 157.4, 106.87) mm, rotated rx -180 ry 0 rz 180 deg; joints [-146.542, -79.523, -29.081, 64.231, 37.75, -58.594]
  MoveL 7560 to (238.49, 157.4, 106.87) mm, rotated rx -180 ry 0 rz 180 deg; joints [-146.542, -79.523, -29.081, 64.231, 37.75, -58.594]
  Call Extruder(264.19935)
  MoveL 7561 to (238.31, 157.7, 106.87) mm, rotated rx 180 ry 0 rz -180 deg; joints [-146.51, -79.527, -29.072, 64.263, 37.775, -58.621]
  MoveL 7562 to (238.31, 157.7, 106.87) mm, rotated rx 180 ry 0 rz -180 deg; joints [-146.51, -79.527, -29.072, 64.263, 37.775, -58.621]
  Call Extruder(264.40786)
  MoveL 7563 to (238.13, 158.01, 106.87) mm, rotated rx -180 ry 0 rz 180 deg; joints [-146.479, -79.532, -29.064, 64.294, 37.8, -58.649]
  MoveL 7564 to (238.13, 158.01, 106.87) mm, rotated rx -180 ry 0 rz 180 deg; joints [-146.479, -79.532, -29.064, 64.294, 37.8, -58.649]
  Call Extruder(264.58740)
  MoveL 7565 to (237.96, 158.25, 106.87) mm, rotated rx 180 ry 0 rz 180 deg; joints [-146.452, -79.529, -29.068, 64.314, 37.824, -58.664]
  MoveL 7566 to (237.96, 158.25, 106.87) mm, rotated rx 180 ry 0 rz 180 deg; joints [-146.452, -79.529, -29.068, 64.314, 37.824, -58.664]
  Call Extruder(264.92080)
  MoveL 7567 to (237.63, 158.7, 106.87) mm, rotated rx 180 ry 0 rz 180 deg; joints [-146.402, -79.525, -29.078, 64.351, 37.869, -58.69]
  MoveL 7568 to (237.63, 158.7, 106.87) mm, rotated rx 180 ry 0 rz 180 deg; joints [-146.402, -79.525, -29.078, 64.351, 37.869, -58.69]
  Call Extruder(265.25540)
  MoveL 7569 to (237.3, 159.15, 106.87) mm, rotated rx -180 ry 0 rz 180 deg; joints [-146.352, -79.52, -29.087, 64.388, 37.913, -58.716]
  Call Extruder(266.08335)
  MoveL 7570 to (236.39, 160.19, 106.87) mm, rotated rx 180 ry 0 rz 180 deg; joints [-146.229, -79.483, -29.162, 64.448, 38.034, -58.743]
  Call Extruder(266.91129)
  MoveL 7571 to (235.35, 161.1, 106.87) mm, rotated rx -180 ry 0 rz 180 deg; joints [-146.109, -79.412, -29.305, 64.466, 38.168, -58.717]
  Call Extruder(267.07860)
  MoveL 7572 to (235.13, 161.27, 106.87) mm, rotated rx 180 ry 0 rz 180 deg; joints [-146.086, -79.392, -29.344, 64.463, 38.196, -58.704]
  MoveL 7573 to (235.13, 161.27, 106.87) mm, rotated rx 180 ry 0 rz 180 deg; joints [-146.086, -79.392, -29.344, 64.463, 38.196, -58.704]
  Call Extruder(267.41202)
  MoveL 7574 to (234.68, 161.59, 106.87) mm, rotated rx -180 ry 0 rz 180 deg; joints [-146.039, -79.354, -29.421, 64.458, 38.253, -58.678]
  MoveL 7575 to (234.68, 161.59, 106.87) mm, rotated rx -180 ry 0 rz 180 deg; joints [-146.039, -79.354, -29.421, 64.458, 38.253, -58.678]
  Call Extruder(267.74426)
  MoveL 7576 to (234.23, 161.92, 106.87) mm, rotated rx -180 ry 0 rz 180 deg; joints [-145.992, -79.316, -29.498, 64.454, 38.31, -58.653]
  MoveL 7577 to (234.23, 161.92, 106.87) mm, rotated rx -180 ry 0 rz 180 deg; joints [-145.992, -79.316, -29.498, 64.454, 38.31, -58.653]
  Call Extruder(267.86192)
  MoveL 7578 to (234.05, 162.02, 106.87) mm, rotated rx -180 ry 0 rz -180 deg; joints [-145.976, -79.298, -29.533, 64.447, 38.331, -58.638]
  MoveL 7579 to (234.05, 162.02, 106.87) mm, rotated rx -180 ry 0 rz -180 deg; joints [-145.976, -79.298, -29.533, 64.447, 38.331, -58.638]
  Call Extruder(268.06964)
  MoveL 7580 to (233.75, 162.2, 106.87) mm, rotated rx 180 ry 0 rz 180 deg; joints [-145.947, -79.268, -29.595, 64.436, 38.369, -58.612]
  MoveL 7581 to (233.75, 162.2, 106.87) mm, rotated rx 180 ry 0 rz 180 deg; joints [-145.947, -79.268, -29.595, 64.436, 38.369, -58.612]
  Call Extruder(268.27659)
  MoveL 7582 to (233.45, 162.37, 106.87) mm, rotated rx 180 ry 0 rz 180 deg; joints [-145.919, -79.237, -29.657, 64.424, 38.407, -58.585]
  MoveL 7583 to (233.45, 162.37, 106.87) mm, rotated rx 180 ry 0 rz 180 deg; joints [-145.919, -79.237, -29.657, 64.424, 38.407, -58.585]
  Call Extruder(268.48276)
  MoveL 7584 to (233.14, 162.55, 106.87) mm, rotated rx 180 ry 0 rz 180 deg; joints [-145.891, -79.206, -29.718, 64.413, 38.444, -58.559]
  MoveL 7585 to (233.14, 162.55, 106.87) mm, rotated rx 180 ry 0 rz 180 deg; joints [-145.891, -79.206, -29.718, 64.413, 38.444, -58.559]
  Call Extruder(268.66443)
  MoveL 7586 to (232.86, 162.69, 106.87) mm, rotated rx 180 ry 0 rz -180 deg; joints [-145.866, -79.177, -29.778, 64.399, 38.478, -58.531]
  MoveL 7587 to (232.86, 162.69, 106.87) mm, rotated rx 180 ry 0 rz -180 deg; joints [-145.866, -79.177, -29.778, 64.399, 38.478, -58.531]
  Call Extruder(268.82240)
  MoveL 7588 to (232.62, 162.8, 106.87) mm, rotated rx 180 ry 0 rz 180 deg; joints [-145.845, -79.148, -29.837, 64.383, 38.508, -58.502]
  MoveL 7589 to (232.62, 162.8, 106.87) mm, rotated rx 180 ry 0 rz 180 deg; joints [-145.845, -79.148, -29.837, 64.383, 38.508, -58.502]
  Call Extruder(268.97977)
  MoveL 7590 to (232.37, 162.9, 106.87) mm, rotated rx 180 ry 0 rz 180 deg; joints [-145.825, -79.119, -29.895, 64.367, 38.539, -58.473]
  MoveL 7591 to (232.37, 162.9, 106.87) mm, rotated rx 180 ry 0 rz 180 deg; joints [-145.825, -79.119, -29.895, 64.367, 38.539, -58.473]
  Call Extruder(269.16252)
  MoveL 7592 to (232.08, 163.03, 106.87) mm, rotated rx 180 ry 0 rz 180 deg; joints [-145.801, -79.084, -29.964, 64.347, 38.574, -58.438]
  MoveL 7593 to (232.08, 163.03, 106.87) mm, rotated rx 180 ry 0 rz 180 deg; joints [-145.801, -79.084, -29.964, 64.347, 38.574, -58.438]
  Call Extruder(269.34450)
  MoveL 7594 to (231.78, 163.15, 106.87) mm, rotated rx -180 ry 0 rz 180 deg; joints [-145.777, -79.05, -30.033, 64.328, 38.609, -58.403]
  MoveL 7595 to (231.78, 163.15, 106.87) mm, rotated rx -180 ry 0 rz 180 deg; joints [-145.777, -79.05, -30.033, 64.328, 38.609, -58.403]
  Call Extruder(269.49184)
  MoveL 7596 to (231.54, 163.24, 106.87) mm, rotated rx 180 ry 0 rz 180 deg; joints [-145.759, -79.021, -30.092, 64.31, 38.638, -58.373]
  MoveL 7597 to (231.54, 163.24, 106.87) mm, rotated rx 180 ry 0 rz 180 deg; joints [-145.759, -79.021, -30.092, 64.31, 38.638, -58.373]
  Call Extruder(269.60506)
  MoveL 7598 to (231.35, 163.3, 106.87) mm, rotated rx -180 ry 0 rz 180 deg; joints [-145.744, -78.997, -30.14, 64.295, 38.661, -58.347]
  MoveL 7599 to (231.35, 163.3, 106.87) mm, rotated rx -180 ry 0 rz 180 deg; joints [-145.744, -78.997, -30.14, 64.295, 38.661, -58.347]
  Call Extruder(269.71784)
  MoveL 7600 to (231.17, 163.36, 106.87) mm, rotated rx 180 ry 0 rz 180 deg; joints [-145.73, -78.973, -30.188, 64.279, 38.683, -58.322]
  MoveL 7601 to (231.17, 163.36, 106.87) mm, rotated rx 180 ry 0 rz 180 deg; joints [-145.73, -78.973, -30.188, 64.279, 38.683, -58.322]
  Call Extruder(269.83017)
  MoveL 7602 to (230.98, 163.42, 106.87) mm, rotated rx 180 ry 0 rz 180 deg; joints [-145.716, -78.949, -30.237, 64.264, 38.706, -58.296]
  MoveL 7603 to (230.98, 163.42, 106.87) mm, rotated rx 180 ry 0 rz 180 deg; joints [-145.716, -78.949, -30.237, 64.264, 38.706, -58.296]
  Call Extruder(269.94206)
  MoveL 7604 to (230.79, 163.48, 106.87) mm, rotated rx 180 ry 0 rz 180 deg; joints [-145.702, -78.925, -30.284, 64.249, 38.728, -58.27]
  MoveL 7605 to (230.79, 163.48, 106.87) mm, rotated rx 180 ry 0 rz 180 deg; joints [-145.702, -78.925, -30.284, 64.249, 38.728, -58.27]
  Call Extruder(270.06346)
  MoveL 7606 to (230.58, 163.55, 106.87) mm, rotated rx -180 ry 0 rz 180 deg; joints [-145.687, -78.899, -30.337, 64.232, 38.753, -58.242]
  MoveL 7607 to (230.58, 163.55, 106.87) mm, rotated rx -180 ry 0 rz 180 deg; joints [-145.687, -78.899, -30.337, 64.232, 38.753, -58.242]
  Call Extruder(270.19428)
  MoveL 7608 to (230.36, 163.61, 106.87) mm, rotated rx 180 ry 0 rz -180 deg; joints [-145.67, -78.87, -30.395, 64.213, 38.78, -58.211]
  MoveL 7609 to (230.36, 163.61, 106.87) mm, rotated rx 180 ry 0 rz -180 deg; joints [-145.67, -78.87, -30.395, 64.213, 38.78, -58.211]
  Call Extruder(270.32452)
  MoveL 7610 to (230.14, 163.68, 106.87) mm, rotated rx -180 ry 0 rz 180 deg; joints [-145.654, -78.842, -30.453, 64.194, 38.806, -58.18]
  MoveL 7611 to (230.14, 163.68, 106.87) mm, rotated rx -180 ry 0 rz 180 deg; joints [-145.654, -78.842, -30.453, 64.194, 38.806, -58.18]
  Call Extruder(270.45421)
  MoveL 7612 to (229.91, 163.75, 106.87) mm, rotated rx 180 ry 0 rz 180 deg; joints [-145.638, -78.813, -30.511, 64.175, 38.833, -58.149]
  MoveL 7613 to (229.91, 163.75, 106.87) mm, rotated rx 180 ry 0 rz 180 deg; joints [-145.638, -78.813, -30.511, 64.175, 38.833, -58.149]
  Call Extruder(270.58333)
  MoveL 7614 to (229.69, 163.82, 106.87) mm, rotated rx -180 ry 0 rz 180 deg; joints [-145.621, -78.784, -30.569, 64.156, 38.859, -58.118]
  MoveL 7615 to (229.69, 163.82, 106.87) mm, rotated rx -180 ry 0 rz 180 deg; joints [-145.621, -78.784, -30.569, 64.156, 38.859, -58.118]
  Call Extruder(270.69840)
  MoveL 7616 to (229.48, 163.86, 106.87) mm, rotated rx -180 ry 0 rz 180 deg; joints [-145.607, -78.756, -30.625, 64.136, 38.883, -58.086]
  MoveL 7617 to (229.48, 163.86, 106.87) mm, rotated rx -180 ry 0 rz 180 deg; joints [-145.607, -78.756, -30.625, 64.136, 38.883, -58.086]
  Call Extruder(270.81302)
  MoveL 7618 to (229.28, 163.91, 106.87) mm, rotated rx 180 ry 0 rz -180 deg; joints [-145.594, -78.728, -30.681, 64.116, 38.907, -58.054]
  MoveL 7619 to (229.28, 163.91, 106.87) mm, rotated rx 180 ry 0 rz -180 deg; joints [-145.594, -78.728, -30.681, 64.116, 38.907, -58.054]
  Call Extruder(270.92719)
  MoveL 7620 to (229.08, 163.95, 106.87) mm, rotated rx -180 ry 0 rz 180 deg; joints [-145.58, -78.701, -30.737, 64.096, 38.931, -58.023]
  MoveL 7621 to (229.08, 163.95, 106.87) mm, rotated rx -180 ry 0 rz 180 deg; joints [-145.58, -78.701, -30.737, 64.096, 38.931, -58.023]
  Call Extruder(271.04091)
  MoveL 7622 to (228.87, 164, 106.87) mm, rotated rx 180 ry 0 rz -180 deg; joints [-145.566, -78.673, -30.793, 64.076, 38.956, -57.991]
  MoveL 7623 to (228.87, 164, 106.87) mm, rotated rx 180 ry 0 rz -180 deg; joints [-145.566, -78.673, -30.793, 64.076, 38.956, -57.991]
  Call Extruder(271.16633)
  MoveL 7624 to (228.65, 164.04, 106.87) mm, rotated rx -180 ry 0 rz 180 deg; joints [-145.551, -78.642, -30.856, 64.054, 38.982, -57.956]
  MoveL 7625 to (228.65, 164.04, 106.87) mm, rotated rx -180 ry 0 rz 180 deg; joints [-145.551, -78.642, -30.856, 64.054, 38.982, -57.956]
  Call Extruder(271.30331)
  MoveL 7626 to (228.4, 164.09, 106.87) mm, rotated rx 180 ry 0 rz 180 deg; joints [-145.535, -78.607, -30.925, 64.029, 39.011, -57.917]
  MoveL 7627 to (228.4, 164.09, 106.87) mm, rotated rx 180 ry 0 rz 180 deg; joints [-145.535, -78.607, -30.925, 64.029, 39.011, -57.917]
  Call Extruder(271.43968)
  MoveL 7628 to (228.15, 164.14, 106.87) mm, rotated rx 180 ry 0 rz 180 deg; joints [-145.518, -78.573, -30.995, 64.004, 39.041, -57.878]
  MoveL 7629 to (228.15, 164.14, 106.87) mm, rotated rx 180 ry 0 rz 180 deg; joints [-145.518, -78.573, -30.995, 64.004, 39.041, -57.878]
  Call Extruder(271.57543)
  MoveL 7630 to (227.9, 164.19, 106.87) mm, rotated rx -180 ry 0 rz 180 deg; joints [-145.502, -78.539, -31.064, 63.979, 39.07, -57.839]
  MoveL 7631 to (227.9, 164.19, 106.87) mm, rotated rx -180 ry 0 rz 180 deg; joints [-145.502, -78.539, -31.064, 63.979, 39.07, -57.839]
  Call Extruder(271.71058)
  MoveL 7632 to (227.65, 164.24, 106.87) mm, rotated rx 180 ry 0 rz 180 deg; joints [-145.485, -78.505, -31.133, 63.955, 39.099, -57.8]
  MoveL 7633 to (227.65, 164.24, 106.87) mm, rotated rx 180 ry 0 rz 180 deg; joints [-145.485, -78.505, -31.133, 63.955, 39.099, -57.8]
  Call Extruder(271.84512)
  MoveL 7634 to (227.4, 164.29, 106.87) mm, rotated rx 180 ry 0 rz 180 deg; joints [-145.469, -78.471, -31.201, 63.93, 39.128, -57.762]
  MoveL 7635 to (227.4, 164.29, 106.87) mm, rotated rx 180 ry 0 rz 180 deg; joints [-145.469, -78.471, -31.201, 63.93, 39.128, -57.762]
  Call Extruder(271.97904)
  MoveL 7636 to (227.15, 164.34, 106.87) mm, rotated rx 180 ry 0 rz 180 deg; joints [-145.453, -78.437, -31.27, 63.906, 39.157, -57.723]
  MoveL 7637 to (227.15, 164.34, 106.87) mm, rotated rx 180 ry 0 rz 180 deg; joints [-145.453, -78.437, -31.27, 63.906, 39.157, -57.723]
  Call Extruder(272.12691)
  MoveL 7638 to (226.87, 164.39, 106.87) mm, rotated rx 180 ry 0 rz -180 deg; joints [-145.435, -78.398, -31.347, 63.878, 39.189, -57.679]
  MoveL 7639 to (226.87, 164.39, 106.87) mm, rotated rx 180 ry 0 rz -180 deg; joints [-145.435, -78.398, -31.347, 63.878, 39.189, -57.679]
  Call Extruder(272.28865)
  MoveL 7640 to (226.57, 164.44, 106.87) mm, rotated rx 180 ry 0 rz 180 deg; joints [-145.415, -78.355, -31.434, 63.846, 39.225, -57.63]
  MoveL 7641 to (226.57, 164.44, 106.87) mm, rotated rx 180 ry 0 rz 180 deg; joints [-145.415, -78.355, -31.434, 63.846, 39.225, -57.63]
  Call Extruder(272.44966)
  MoveL 7642 to (226.26, 164.49, 106.87) mm, rotated rx -180 ry 0 rz 180 deg; joints [-145.396, -78.312, -31.521, 63.815, 39.261, -57.58]
  MoveL 7643 to (226.26, 164.49, 106.87) mm, rotated rx -180 ry 0 rz 180 deg; joints [-145.396, -78.312, -31.521, 63.815, 39.261, -57.58]
  Call Extruder(272.60995)
  MoveL 7644 to (225.96, 164.53, 106.87) mm, rotated rx 180 ry 0 rz 180 deg; joints [-145.377, -78.27, -31.607, 63.783, 39.296, -57.531]
  MoveL 7645 to (225.96, 164.53, 106.87) mm, rotated rx 180 ry 0 rz 180 deg; joints [-145.377, -78.27, -31.607, 63.783, 39.296, -57.531]
  Call Extruder(272.76951)
  MoveL 7646 to (225.65, 164.58, 106.87) mm, rotated rx -180 ry 0 rz -180 deg; joints [-145.357, -78.227, -31.693, 63.752, 39.332, -57.483]
  MoveL 7647 to (225.65, 164.58, 106.87) mm, rotated rx -180 ry 0 rz -180 deg; joints [-145.357, -78.227, -31.693, 63.752, 39.332, -57.483]
  Call Extruder(272.92834)
  MoveL 7648 to (225.34, 164.63, 106.87) mm, rotated rx 180 ry 0 rz 180 deg; joints [-145.338, -78.185, -31.779, 63.721, 39.367, -57.434]
  MoveL 7649 to (225.34, 164.63, 106.87) mm, rotated rx 180 ry 0 rz 180 deg; joints [-145.338, -78.185, -31.779, 63.721, 39.367, -57.434]
  Call Extruder(273.10701)
  MoveL 7650 to (225, 164.68, 106.87) mm, rotated rx -180 ry 0 rz 180 deg; joints [-145.317, -78.136, -31.878, 63.685, 39.407, -57.377]
  MoveL 7651 to (225, 164.68, 106.87) mm, rotated rx -180 ry 0 rz 180 deg; joints [-145.317, -78.136, -31.878, 63.685, 39.407, -57.377]
  Call Extruder(273.30545)
  MoveL 7652 to (224.61, 164.72, 106.87) mm, rotated rx -180 ry 0 rz 180 deg; joints [-145.293, -78.081, -31.989, 63.643, 39.452, -57.313]
  MoveL 7653 to (224.61, 164.72, 106.87) mm, rotated rx -180 ry 0 rz 180 deg; joints [-145.293, -78.081, -31.989, 63.643, 39.452, -57.313]
  Call Extruder(273.50302)
  MoveL 7654 to (224.22, 164.77, 106.87) mm, rotated rx -180 ry 0 rz 180 deg; joints [-145.27, -78.026, -32.101, 63.602, 39.497, -57.249]
  MoveL 7655 to (224.22, 164.77, 106.87) mm, rotated rx -180 ry 0 rz 180 deg; joints [-145.27, -78.026, -32.101, 63.602, 39.497, -57.249]
  Call Extruder(273.69973)
  MoveL 7656 to (223.84, 164.82, 106.87) mm, rotated rx 180 ry 0 rz 180 deg; joints [-145.246, -77.971, -32.211, 63.561, 39.542, -57.186]
  MoveL 7657 to (223.84, 164.82, 106.87) mm, rotated rx 180 ry 0 rz 180 deg; joints [-145.246, -77.971, -32.211, 63.561, 39.542, -57.186]
  Call Extruder(273.89557)
  MoveL 7658 to (223.45, 164.86, 106.87) mm, rotated rx 180 ry 0 rz 180 deg; joints [-145.223, -77.916, -32.323, 63.52, 39.586, -57.122]
  MoveL 7659 to (223.45, 164.86, 106.87) mm, rotated rx 180 ry 0 rz 180 deg; joints [-145.223, -77.916, -32.323, 63.52, 39.586, -57.122]
  Call Extruder(274.19092)
  MoveL 7660 to (222.86, 164.91, 106.87) mm, rotated rx -180 ry 0 rz 180 deg; joints [-145.189, -77.83, -32.495, 63.455, 39.654, -57.022]
  MoveL 7661 to (222.86, 164.91, 106.87) mm, rotated rx -180 ry 0 rz 180 deg; joints [-145.189, -77.83, -32.495, 63.455, 39.654, -57.022]
  Call Extruder(274.48494)
  MoveL 7662 to (222.27, 164.96, 106.87) mm, rotated rx 180 ry 0 rz 180 deg; joints [-145.155, -77.745, -32.667, 63.39, 39.721, -56.922]
  MoveL 7663 to (222.27, 164.96, 106.87) mm, rotated rx 180 ry 0 rz 180 deg; joints [-145.155, -77.745, -32.667, 63.39, 39.721, -56.922]
  Call Extruder(274.77764)
  MoveL 7664 to (221.68, 165, 106.87) mm, rotated rx 180 ry 0 rz 180 deg; joints [-145.121, -77.661, -32.839, 63.326, 39.789, -56.824]
  MoveL 7665 to (221.68, 165, 106.87) mm, rotated rx 180 ry 0 rz 180 deg; joints [-145.121, -77.661, -32.839, 63.326, 39.789, -56.824]
  Call Extruder(275.35108)
  MoveL 7666 to (220.52, 165.05, 106.87) mm, rotated rx 180 ry 0 rz 180 deg; joints [-145.056, -77.49, -33.185, 63.193, 39.921, -56.621]
  MoveL 7667 to (220.52, 165.05, 106.87) mm, rotated rx 180 ry 0 rz 180 deg; joints [-145.056, -77.49, -33.185, 63.193, 39.921, -56.621]
  Call Extruder(276.06510)
  MoveL 7668 to (219.06, 165.09, 106.87) mm, rotated rx 180 ry 0 rz 180 deg; joints [-144.977, -77.277, -33.617, 63.028, 40.086, -56.369]
  Call Extruder(392.91185)
  MoveL 7669 to (-19.06, 165.09, 106.87) mm, rotated rx 180 ry 0 rz -180 deg; joints [-127.435, -56.551, -78.268, 61.649, 64.458, -38.627]
  Call Extruder(393.34045)
  MoveL 7670 to (-19.94, 165.07, 106.87) mm, rotated rx -180 ry 0 rz -180 deg; joints [-127.348, -56.505, -78.377, 61.697, 64.542, -38.598]
  MoveL 7671 to (-19.94, 165.07, 106.87) mm, rotated rx -180 ry 0 rz -180 deg; joints [-127.348, -56.505, -78.377, 61.697, 64.542, -38.598]
  Call Extruder(393.91390)
  MoveL 7672 to (-21.1, 165.02, 106.87) mm, rotated rx 180 ry 0 rz 180 deg; joints [-127.235, -56.443, -78.525, 61.76, 64.653, -38.557]
  MoveL 7673 to (-21.1, 165.02, 106.87) mm, rotated rx 180 ry 0 rz 180 deg; joints [-127.235, -56.443, -78.525, 61.76, 64.653, -38.557]
  Call Extruder(394.34820)
  MoveL 7674 to (-21.97, 164.98, 106.87) mm, rotated rx 180 ry 0 rz 180 deg; joints [-127.15, -56.395, -78.638, 61.807, 64.737, -38.525]
  MoveL 7675 to (-21.97, 164.98, 106.87) mm, rotated rx 180 ry 0 rz 180 deg; joints [-127.15, -56.395, -78.638, 61.807, 64.737, -38.525]
  Call Extruder(394.64223)
  MoveL 7676 to (-22.56, 164.93, 106.87) mm, rotated rx 180 ry 0 rz -180 deg; joints [-127.093, -56.362, -78.716, 61.836, 64.793, -38.502]
  MoveL 7677 to (-22.56, 164.93, 106.87) mm, rotated rx 180 ry 0 rz -180 deg; joints [-127.093, -56.362, -78.716, 61.836, 64.793, -38.502]
  Call Extruder(394.93759)
  MoveL 7678 to (-23.15, 164.89, 106.87) mm, rotated rx 180 ry 0 rz 180 deg; joints [-127.037, -56.329, -78.794, 61.866, 64.849, -38.478]
  MoveL 7679 to (-23.15, 164.89, 106.87) mm, rotated rx 180 ry 0 rz 180 deg; joints [-127.037, -56.329, -78.794, 61.866, 64.849, -38.478]
  Call Extruder(395.18380)
  MoveL 7680 to (-23.64, 164.84, 106.87) mm, rotated rx 180 ry 0 rz 180 deg; joints [-126.991, -56.301, -78.86, 61.89, 64.896, -38.458]
  MoveL 7681 to (-23.64, 164.84, 106.87) mm, rotated rx 180 ry 0 rz 180 deg; joints [-126.991, -56.301, -78.86, 61.89, 64.896, -38.458]
  Call Extruder(395.38051)
  MoveL 7682 to (-24.03, 164.79, 106.87) mm, rotated rx 180 ry 0 rz 180 deg; joints [-126.955, -56.279, -78.914, 61.909, 64.933, -38.441]
  MoveL 7683 to (-24.03, 164.79, 106.87) mm, rotated rx 180 ry 0 rz 180 deg; joints [-126.955, -56.279, -78.914, 61.909, 64.933, -38.441]
  Call Extruder(395.57808)
  MoveL 7684 to (-24.42, 164.75, 106.87) mm, rotated rx 180 ry 0 rz -180 deg; joints [-126.919, -56.256, -78.967, 61.927, 64.97, -38.424]
  MoveL 7685 to (-24.42, 164.75, 106.87) mm, rotated rx 180 ry 0 rz -180 deg; joints [-126.919, -56.256, -78.967, 61.927, 64.97, -38.424]
  Call Extruder(395.77652)
  MoveL 7686 to (-24.8, 164.7, 106.87) mm, rotated rx -180 ry 0 rz 180 deg; joints [-126.883, -56.233, -79.021, 61.945, 65.007, -38.407]
  MoveL 7687 to (-24.8, 164.7, 106.87) mm, rotated rx -180 ry 0 rz 180 deg; joints [-126.883, -56.233, -79.021, 61.945, 65.007, -38.407]
  Call Extruder(395.97583)
  MoveL 7688 to (-25.19, 164.66, 106.87) mm, rotated rx -180 ry 0 rz 180 deg; joints [-126.847, -56.211, -79.074, 61.964, 65.044, -38.39]
  MoveL 7689 to (-25.19, 164.66, 106.87) mm, rotated rx -180 ry 0 rz 180 deg; joints [-126.847, -56.211, -79.074, 61.964, 65.044, -38.39]
  Call Extruder(396.13466)
  MoveL 7690 to (-25.5, 164.61, 106.87) mm, rotated rx 180 ry 0 rz 180 deg; joints [-126.82, -56.192, -79.118, 61.977, 65.073, -38.376]
  MoveL 7691 to (-25.5, 164.61, 106.87) mm, rotated rx 180 ry 0 rz 180 deg; joints [-126.82, -56.192, -79.118, 61.977, 65.073, -38.376]
  Call Extruder(396.29423)
  MoveL 7692 to (-25.8, 164.56, 106.87) mm, rotated rx 180 ry 0 rz 180 deg; joints [-126.792, -56.174, -79.162, 61.99, 65.102, -38.361]
  MoveL 7693 to (-25.8, 164.56, 106.87) mm, rotated rx 180 ry 0 rz 180 deg; joints [-126.792, -56.174, -79.162, 61.99, 65.102, -38.361]
  Call Extruder(396.45451)
  MoveL 7694 to (-26.11, 164.51, 106.87) mm, rotated rx -180 ry 0 rz 180 deg; joints [-126.765, -56.155, -79.206, 62.004, 65.131, -38.346]
  MoveL 7695 to (-26.11, 164.51, 106.87) mm, rotated rx -180 ry 0 rz 180 deg; joints [-126.765, -56.155, -79.206, 62.004, 65.131, -38.346]
  Call Extruder(396.61553)
  MoveL 7696 to (-26.41, 164.46, 106.87) mm, rotated rx -180 ry 0 rz 180 deg; joints [-126.737, -56.137, -79.25, 62.017, 65.16, -38.331]
  MoveL 7697 to (-26.41, 164.46, 106.87) mm, rotated rx -180 ry 0 rz 180 deg; joints [-126.737, -56.137, -79.25, 62.017, 65.16, -38.331]
  Call Extruder(396.77727)
  MoveL 7698 to (-26.72, 164.41, 106.87) mm, rotated rx 180 ry 0 rz 180 deg; joints [-126.71, -56.118, -79.294, 62.031, 65.189, -38.317]
  MoveL 7699 to (-26.72, 164.41, 106.87) mm, rotated rx 180 ry 0 rz 180 deg; joints [-126.71, -56.118, -79.294, 62.031, 65.189, -38.317]
  Call Extruder(396.93974)
  MoveL 7700 to (-27.03, 164.37, 106.87) mm, rotated rx 180 ry 0 rz 180 deg; joints [-126.682, -56.1, -79.338, 62.044, 65.218, -38.302]
  MoveL 7701 to (-27.03, 164.37, 106.87) mm, rotated rx 180 ry 0 rz 180 deg; joints [-126.682, -56.1, -79.338, 62.044, 65.218, -38.302]
  Call Extruder(397.07367)
  MoveL 7702 to (-27.27, 164.32, 106.87) mm, rotated rx 180 ry 0 rz 180 deg; joints [-126.66, -56.084, -79.375, 62.054, 65.242, -38.289]
  MoveL 7703 to (-27.27, 164.32, 106.87) mm, rotated rx 180 ry 0 rz 180 deg; joints [-126.66, -56.084, -79.375, 62.054, 65.242, -38.289]
  Call Extruder(397.20821)
  MoveL 7704 to (-27.52, 164.27, 106.87) mm, rotated rx 180 ry 0 rz 180 deg; joints [-126.638, -56.068, -79.413, 62.064, 65.265, -38.275]
  MoveL 7705 to (-27.52, 164.27, 106.87) mm, rotated rx 180 ry 0 rz 180 deg; joints [-126.638, -56.068, -79.413, 62.064, 65.265, -38.275]
  Call Extruder(397.34335)
  MoveL 7706 to (-27.77, 164.22, 106.87) mm, rotated rx -180 ry 0 rz -180 deg; joints [-126.617, -56.053, -79.45, 62.074, 65.289, -38.262]
  MoveL 7707 to (-27.77, 164.22, 106.87) mm, rotated rx -180 ry 0 rz -180 deg; joints [-126.617, -56.053, -79.45, 62.074, 65.289, -38.262]
  Call Extruder(397.47911)
  MoveL 7708 to (-28.02, 164.17, 106.87) mm, rotated rx -180 ry 0 rz 180 deg; joints [-126.595, -56.037, -79.487, 62.084, 65.312, -38.249]
  MoveL 7709 to (-28.02, 164.17, 106.87) mm, rotated rx -180 ry 0 rz 180 deg; joints [-126.595, -56.037, -79.487, 62.084, 65.312, -38.249]
  Call Extruder(397.61548)
  MoveL 7710 to (-28.27, 164.12, 106.87) mm, rotated rx -180 ry 0 rz 180 deg; joints [-126.573, -56.021, -79.524, 62.094, 65.336, -38.236]
  MoveL 7711 to (-28.27, 164.12, 106.87) mm, rotated rx -180 ry 0 rz 180 deg; joints [-126.573, -56.021, -79.524, 62.094, 65.336, -38.236]
  Call Extruder(397.70034)
  MoveL 7712 to (-28.43, 164.09, 106.87) mm, rotated rx 180 ry 0 rz 180 deg; joints [-126.559, -56.012, -79.547, 62.101, 65.351, -38.228]
  Set speed (130.0 mm/s)
  MoveL 7713 to (-31.76, 163.31, 106.87) mm, rotated rx 180 ry 0 rz 180 deg; joints [-126.274, -55.796, -80.061, 62.227, 65.666, -38.041]
  MoveL 7714 to (-31.76, 163.31, 116.27) mm, rotated rx 180 ry 0 rz -180 deg; joints [-126.274, -54.543, -80.572, 62.527, 65.322, -38.764]
  Call Extruder(395.70034)
  Set speed (40.0 mm/s)
  MoveL 7715 to (-31.76, 163.31, 116.27) mm, rotated rx 180 ry 0 rz -180 deg; joints [-126.274, -54.543, -80.572, 62.527, 65.322, -38.764]
  Call Extruder(0.00000)
  Set speed (130.0 mm/s)
  MoveL 7716 to (-34.22, 161.92, 116.27) mm, rotated rx -180 ry 0 rz 180 deg; joints [-126.122, -54.327, -81.077, 62.54, 65.55, -38.535]
  Call Extruder(2.00000)
  Set speed (40.0 mm/s)
  MoveL 7717 to (-34.22, 161.92, 116.27) mm, rotated rx -180 ry 0 rz 180 deg; joints [-126.122, -54.327, -81.077, 62.54, 65.55, -38.535]
  Set speed (30.0 mm/s)
  MoveL 7718 to (-34.22, 161.92, 116.27) mm, rotated rx -180 ry 0 rz 180 deg; joints [-126.122, -54.327, -81.077, 62.54, 65.55, -38.535]
  Call Extruder(2.16612)
  MoveL 7719 to (-34.45, 161.76, 116.27) mm, rotated rx -180 ry 0 rz 180 deg; joints [-126.111, -54.305, -81.13, 62.537, 65.571, -38.51]
  MoveL 7720 to (-34.45, 161.76, 116.27) mm, rotated rx -180 ry 0 rz 180 deg; joints [-126.111, -54.305, -81.13, 62.537, 65.571, -38.51]
  Call Extruder(2.49954)
  MoveL 7721 to (-34.9, 161.43, 116.27) mm, rotated rx -180 ry 0 rz 180 deg; joints [-126.089, -54.26, -81.233, 62.533, 65.612, -38.46]
  MoveL 7722 to (-34.9, 161.43, 116.27) mm, rotated rx -180 ry 0 rz 180 deg; joints [-126.089, -54.26, -81.233, 62.533, 65.612, -38.46]
  Call Extruder(2.83415)
  MoveL 7723 to (-35.35, 161.1, 116.27) mm, rotated rx 180 ry 0 rz 180 deg; joints [-126.067, -54.216, -81.337, 62.528, 65.654, -38.41]
  Call Extruder(3.66207)
  MoveL 7724 to (-36.39, 160.19, 116.27) mm, rotated rx 180 ry 0 rz 180 deg; joints [-126.027, -54.104, -81.6, 62.501, 65.748, -38.277]
  Call Extruder(4.49000)
  MoveL 7725 to (-37.3, 159.15, 116.27) mm, rotated rx 180 ry 0 rz 180 deg; joints [-126.011, -53.99, -81.868, 62.454, 65.829, -38.133]
  Call Extruder(4.65731)
  MoveL 7726 to (-37.47, 158.93, 116.27) mm, rotated rx -180 ry 0 rz 180 deg; joints [-126.011, -53.967, -81.923, 62.442, 65.844, -38.102]
  MoveL 7727 to (-37.47, 158.93, 116.27) mm, rotated rx -180 ry 0 rz 180 deg; joints [-126.011, -53.967, -81.923, 62.442, 65.844, -38.102]
  Call Extruder(4.99074)
  MoveL 7728 to (-37.79, 158.48, 116.27) mm, rotated rx 180 ry 0 rz 180 deg; joints [-126.011, -53.921, -82.031, 62.417, 65.873, -38.041]
  MoveL 7729 to (-37.79, 158.48, 116.27) mm, rotated rx 180 ry 0 rz 180 deg; joints [-126.011, -53.921, -82.031, 62.417, 65.873, -38.041]
  Call Extruder(5.32299)
  MoveL 7730 to (-38.12, 158.02, 116.27) mm, rotated rx -180 ry 0 rz 180 deg; joints [-126.011, -53.876, -82.14, 62.392, 65.902, -37.981]
  MoveL 7731 to (-38.12, 158.02, 116.27) mm, rotated rx -180 ry 0 rz 180 deg; joints [-126.011, -53.876, -82.14, 62.392, 65.902, -37.981]
  Call Extruder(5.44066)
  MoveL 7732 to (-38.22, 157.85, 116.27) mm, rotated rx 180 ry 0 rz 180 deg; joints [-126.013, -53.859, -82.178, 62.381, 65.91, -37.958]
  MoveL 7733 to (-38.22, 157.85, 116.27) mm, rotated rx 180 ry 0 rz 180 deg; joints [-126.013, -53.859, -82.178, 62.381, 65.91, -37.958]
  Call Extruder(5.64838)
  MoveL 7734 to (-38.4, 157.55, 116.27) mm, rotated rx 180 ry 0 rz 180 deg; joints [-126.018, -53.831, -82.245, 62.361, 65.925, -37.919]
  MoveL 7735 to (-38.4, 157.55, 116.27) mm, rotated rx 180 ry 0 rz 180 deg; joints [-126.018, -53.831, -82.245, 62.361, 65.925, -37.919]
  Call Extruder(5.85533)
  MoveL 7736 to (-38.57, 157.25, 116.27) mm, rotated rx -180 ry 0 rz -180 deg; joints [-126.023, -53.802, -82.313, 62.342, 65.941, -37.879]
  MoveL 7737 to (-38.57, 157.25, 116.27) mm, rotated rx -180 ry 0 rz -180 deg; joints [-126.023, -53.802, -82.313, 62.342, 65.941, -37.879]
  Call Extruder(6.06150)
  MoveL 7738 to (-38.75, 156.94, 116.27) mm, rotated rx 180 ry 0 rz 180 deg; joints [-126.028, -53.773, -82.381, 62.322, 65.956, -37.84]
  MoveL 7739 to (-38.75, 156.94, 116.27) mm, rotated rx 180 ry 0 rz 180 deg; joints [-126.028, -53.773, -82.381, 62.322, 65.956, -37.84]
  Call Extruder(6.24318)
  MoveL 7740 to (-38.89, 156.67, 116.27) mm, rotated rx 180 ry 0 rz 180 deg; joints [-126.034, -53.748, -82.44, 62.303, 65.968, -37.804]
  MoveL 7741 to (-38.89, 156.67, 116.27) mm, rotated rx 180 ry 0 rz 180 deg; joints [-126.034, -53.748, -82.44, 62.303, 65.968, -37.804]
  Call Extruder(6.40116)
  MoveL 7742 to (-39, 156.42, 116.27) mm, rotated rx 180 ry 0 rz 180 deg; joints [-126.042, -53.727, -82.491, 62.284, 65.977, -37.773]
  MoveL 7743 to (-39, 156.42, 116.27) mm, rotated rx 180 ry 0 rz 180 deg; joints [-126.042, -53.727, -82.491, 62.284, 65.977, -37.773]
  Call Extruder(6.55855)
  MoveL 7744 to (-39.1, 156.17, 116.27) mm, rotated rx 180 ry 0 rz -180 deg; joints [-126.05, -53.705, -82.543, 62.266, 65.986, -37.741]
  MoveL 7745 to (-39.1, 156.17, 116.27) mm, rotated rx 180 ry 0 rz -180 deg; joints [-126.05, -53.705, -82.543, 62.266, 65.986, -37.741]
  Call Extruder(6.74127)
  MoveL 7746 to (-39.22, 155.88, 116.27) mm, rotated rx 180 ry 0 rz 180 deg; joints [-126.06, -53.68, -82.602, 62.244, 65.995, -37.705]
  MoveL 7747 to (-39.22, 155.88, 116.27) mm, rotated rx 180 ry 0 rz 180 deg; joints [-126.06, -53.68, -82.602, 62.244, 65.995, -37.705]
  Call Extruder(6.92323)
  MoveL 7748 to (-39.35, 155.58, 116.27) mm, rotated rx 180 ry 0 rz 180 deg; joints [-126.07, -53.655, -82.661, 62.222, 66.005, -37.668]
  MoveL 7749 to (-39.35, 155.58, 116.27) mm, rotated rx 180 ry 0 rz 180 deg; joints [-126.07, -53.655, -82.661, 62.222, 66.005, -37.668]
  Call Extruder(7.07056)
  MoveL 7750 to (-39.44, 155.34, 116.27) mm, rotated rx 180 ry 0 rz 180 deg; joints [-126.079, -53.635, -82.709, 62.203, 66.013, -37.638]
  MoveL 7751 to (-39.44, 155.34, 116.27) mm, rotated rx 180 ry 0 rz 180 deg; joints [-126.079, -53.635, -82.709, 62.203, 66.013, -37.638]
  Call Extruder(7.18380)
  MoveL 7752 to (-39.5, 155.15, 116.27) mm, rotated rx 180 ry 0 rz 180 deg; joints [-126.087, -53.619, -82.746, 62.188, 66.018, -37.615]
  MoveL 7753 to (-39.5, 155.15, 116.27) mm, rotated rx 180 ry 0 rz 180 deg; joints [-126.087, -53.619, -82.746, 62.188, 66.018, -37.615]
  Call Extruder(7.29659)
  MoveL 7754 to (-39.56, 154.97, 116.27) mm, rotated rx 180 ry 0 rz 180 deg; joints [-126.095, -53.604, -82.782, 62.173, 66.023, -37.591]
  MoveL 7755 to (-39.56, 154.97, 116.27) mm, rotated rx 180 ry 0 rz 180 deg; joints [-126.095, -53.604, -82.782, 62.173, 66.023, -37.591]
  Call Extruder(7.40893)
  MoveL 7756 to (-39.62, 154.78, 116.27) mm, rotated rx -180 ry 0 rz 180 deg; joints [-126.103, -53.589, -82.818, 62.157, 66.027, -37.568]
  MoveL 7757 to (-39.62, 154.78, 116.27) mm, rotated rx -180 ry 0 rz 180 deg; joints [-126.103, -53.589, -82.818, 62.157, 66.027, -37.568]
  Call Extruder(7.52083)
  MoveL 7758 to (-39.68, 154.59, 116.27) mm, rotated rx 180 ry 0 rz 180 deg; joints [-126.111, -53.573, -82.855, 62.142, 66.032, -37.545]
  MoveL 7759 to (-39.68, 154.59, 116.27) mm, rotated rx 180 ry 0 rz 180 deg; joints [-126.111, -53.573, -82.855, 62.142, 66.032, -37.545]
  Call Extruder(7.64223)
  MoveL 7760 to (-39.75, 154.38, 116.27) mm, rotated rx 180 ry 0 rz -180 deg; joints [-126.12, -53.557, -82.894, 62.125, 66.037, -37.52]
  MoveL 7761 to (-39.75, 154.38, 116.27) mm, rotated rx 180 ry 0 rz -180 deg; joints [-126.12, -53.557, -82.894, 62.125, 66.037, -37.52]
  Call Extruder(7.77303)
  MoveL 7762 to (-39.81, 154.16, 116.27) mm, rotated rx 180 ry 0 rz 180 deg; joints [-126.131, -53.539, -82.937, 62.106, 66.043, -37.492]
  MoveL 7763 to (-39.81, 154.16, 116.27) mm, rotated rx 180 ry 0 rz 180 deg; joints [-126.131, -53.539, -82.937, 62.106, 66.043, -37.492]
  Call Extruder(7.90326)
  MoveL 7764 to (-39.88, 153.94, 116.27) mm, rotated rx 180 ry 0 rz 180 deg; joints [-126.141, -53.521, -82.979, 62.088, 66.048, -37.465]
  MoveL 7765 to (-39.88, 153.94, 116.27) mm, rotated rx 180 ry 0 rz 180 deg; joints [-126.141, -53.521, -82.979, 62.088, 66.048, -37.465]
  Call Extruder(8.03292)
  MoveL 7766 to (-39.95, 153.71, 116.27) mm, rotated rx 180 ry 0 rz -180 deg; joints [-126.151, -53.503, -83.022, 62.069, 66.053, -37.437]
  MoveL 7767 to (-39.95, 153.71, 116.27) mm, rotated rx 180 ry 0 rz -180 deg; joints [-126.151, -53.503, -83.022, 62.069, 66.053, -37.437]
  Call Extruder(8.16202)
  MoveL 7768 to (-40.02, 153.49, 116.27) mm, rotated rx -180 ry 0 rz 180 deg; joints [-126.161, -53.485, -83.064, 62.051, 66.058, -37.41]
  MoveL 7769 to (-40.02, 153.49, 116.27) mm, rotated rx -180 ry 0 rz 180 deg; joints [-126.161, -53.485, -83.064, 62.051, 66.058, -37.41]
  Call Extruder(8.27711)
  MoveL 7770 to (-40.06, 153.28, 116.27) mm, rotated rx -180 ry 0 rz 180 deg; joints [-126.173, -53.47, -83.101, 62.033, 66.062, -37.386]
  MoveL 7771 to (-40.06, 153.28, 116.27) mm, rotated rx -180 ry 0 rz 180 deg; joints [-126.173, -53.47, -83.101, 62.033, 66.062, -37.386]
  Call Extruder(8.39175)
  MoveL 7772 to (-40.11, 153.08, 116.27) mm, rotated rx -180 ry 0 rz 180 deg; joints [-126.184, -53.454, -83.138, 62.014, 66.065, -37.361]
  MoveL 7773 to (-40.11, 153.08, 116.27) mm, rotated rx -180 ry 0 rz 180 deg; joints [-126.184, -53.454, -83.138, 62.014, 66.065, -37.361]
  Call Extruder(8.50593)
  MoveL 7774 to (-40.15, 152.88, 116.27) mm, rotated rx 180 ry 0 rz 180 deg; joints [-126.195, -53.439, -83.174, 61.996, 66.068, -37.336]
  MoveL 7775 to (-40.15, 152.88, 116.27) mm, rotated rx 180 ry 0 rz 180 deg; joints [-126.195, -53.439, -83.174, 61.996, 66.068, -37.336]
  Call Extruder(8.61966)
  MoveL 7776 to (-40.2, 152.67, 116.27) mm, rotated rx 180 ry 0 rz 180 deg; joints [-126.206, -53.423, -83.211, 61.978, 66.071, -37.312]
  MoveL 7777 to (-40.2, 152.67, 116.27) mm, rotated rx 180 ry 0 rz 180 deg; joints [-126.206, -53.423, -83.211, 61.978, 66.071, -37.312]
  Call Extruder(8.74509)
  MoveL 7778 to (-40.24, 152.44, 116.27) mm, rotated rx 180 ry 0 rz 180 deg; joints [-126.219, -53.406, -83.252, 61.958, 66.075, -37.285]
  MoveL 7779 to (-40.24, 152.44, 116.27) mm, rotated rx 180 ry 0 rz 180 deg; joints [-126.219, -53.406, -83.252, 61.958, 66.075, -37.285]
  Call Extruder(8.88206)
  MoveL 7780 to (-40.29, 152.19, 116.27) mm, rotated rx 180 ry 0 rz 180 deg; joints [-126.233, -53.388, -83.296, 61.935, 66.078, -37.255]
  MoveL 7781 to (-40.29, 152.19, 116.27) mm, rotated rx 180 ry 0 rz 180 deg; joints [-126.233, -53.388, -83.296, 61.935, 66.078, -37.255]
  Call Extruder(9.01843)
  MoveL 7782 to (-40.34, 151.95, 116.27) mm, rotated rx 180 ry 0 rz 180 deg; joints [-126.248, -53.369, -83.34, 61.913, 66.081, -37.225]
  MoveL 7783 to (-40.34, 151.95, 116.27) mm, rotated rx 180 ry 0 rz 180 deg; joints [-126.248, -53.369, -83.34, 61.913, 66.081, -37.225]
  Call Extruder(9.15418)
  MoveL 7784 to (-40.39, 151.7, 116.27) mm, rotated rx 180 ry 0 rz 180 deg; joints [-126.262, -53.35, -83.384, 61.89, 66.085, -37.195]
  MoveL 7785 to (-40.39, 151.7, 116.27) mm, rotated rx 180 ry 0 rz 180 deg; joints [-126.262, -53.35, -83.384, 61.89, 66.085, -37.195]
  Call Extruder(9.28933)
  MoveL 7786 to (-40.44, 151.45, 116.27) mm, rotated rx 180 ry 0 rz -180 deg; joints [-126.276, -53.332, -83.429, 61.868, 66.088, -37.165]
  MoveL 7787 to (-40.44, 151.45, 116.27) mm, rotated rx 180 ry 0 rz -180 deg; joints [-126.276, -53.332, -83.429, 61.868, 66.088, -37.165]
  Call Extruder(9.42386)
  MoveL 7788 to (-40.49, 151.2, 116.27) mm, rotated rx 180 ry 0 rz 180 deg; joints [-126.291, -53.313, -83.473, 61.845, 66.092, -37.136]
  MoveL 7789 to (-40.49, 151.2, 116.27) mm, rotated rx 180 ry 0 rz 180 deg; joints [-126.291, -53.313, -83.473, 61.845, 66.092, -37.136]
  Call Extruder(9.55779)
  MoveL 7790 to (-40.54, 150.95, 116.27) mm, rotated rx 180 ry 0 rz 180 deg; joints [-126.305, -53.295, -83.517, 61.823, 66.095, -37.106]
  MoveL 7791 to (-40.54, 150.95, 116.27) mm, rotated rx 180 ry 0 rz 180 deg; joints [-126.305, -53.295, -83.517, 61.823, 66.095, -37.106]
  Call Extruder(9.70564)
  MoveL 7792 to (-40.59, 150.67, 116.27) mm, rotated rx -180 ry 0 rz 180 deg; joints [-126.322, -53.275, -83.565, 61.797, 66.098, -37.073]
  MoveL 7793 to (-40.59, 150.67, 116.27) mm, rotated rx -180 ry 0 rz 180 deg; joints [-126.322, -53.275, -83.565, 61.797, 66.098, -37.073]
  Call Extruder(9.86737)
  MoveL 7794 to (-40.64, 150.37, 116.27) mm, rotated rx -180 ry 0 rz -180 deg; joints [-126.341, -53.252, -83.618, 61.769, 66.101, -37.037]
  MoveL 7795 to (-40.64, 150.37, 116.27) mm, rotated rx -180 ry 0 rz -180 deg; joints [-126.341, -53.252, -83.618, 61.769, 66.101, -37.037]
  Call Extruder(10.02836)
  MoveL 7796 to (-40.69, 150.06, 116.27) mm, rotated rx 180 ry 0 rz 180 deg; joints [-126.36, -53.23, -83.671, 61.74, 66.104, -37]
  MoveL 7797 to (-40.69, 150.06, 116.27) mm, rotated rx 180 ry 0 rz 180 deg; joints [-126.36, -53.23, -83.671, 61.74, 66.104, -37]
  Call Extruder(10.18863)
  MoveL 7798 to (-40.74, 149.76, 116.27) mm, rotated rx 180 ry 0 rz 180 deg; joints [-126.379, -53.208, -83.723, 61.712, 66.107, -36.964]
  MoveL 7799 to (-40.74, 149.76, 116.27) mm, rotated rx 180 ry 0 rz 180 deg; joints [-126.379, -53.208, -83.723, 61.712, 66.107, -36.964]
  Call Extruder(10.34817)
  MoveL 7800 to (-40.78, 149.45, 116.27) mm, rotated rx 180 ry 0 rz -180 deg; joints [-126.398, -53.186, -83.776, 61.683, 66.11, -36.928]
  MoveL 7801 to (-40.78, 149.45, 116.27) mm, rotated rx 180 ry 0 rz -180 deg; joints [-126.398, -53.186, -83.776, 61.683, 66.11, -36.928]
  Call Extruder(10.50698)
  MoveL 7802 to (-40.83, 149.14, 116.27) mm, rotated rx -180 ry 0 rz 180 deg; joints [-126.417, -53.164, -83.829, 61.655, 66.114, -36.892]
  MoveL 7803 to (-40.83, 149.14, 116.27) mm, rotated rx -180 ry 0 rz 180 deg; joints [-126.417, -53.164, -83.829, 61.655, 66.114, -36.892]
  Call Extruder(10.68565)
  MoveL 7804 to (-40.88, 148.8, 116.27) mm, rotated rx -180 ry 0 rz 180 deg; joints [-126.439, -53.14, -83.887, 61.622, 66.116, -36.851]
  MoveL 7805 to (-40.88, 148.8, 116.27) mm, rotated rx -180 ry 0 rz 180 deg; joints [-126.439, -53.14, -83.887, 61.622, 66.116, -36.851]
  Call Extruder(10.88409)
  MoveL 7806 to (-40.92, 148.41, 116.27) mm, rotated rx 180 ry 0 rz 180 deg; joints [-126.465, -53.113, -83.952, 61.584, 66.119, -36.806]
  MoveL 7807 to (-40.92, 148.41, 116.27) mm, rotated rx 180 ry 0 rz 180 deg; joints [-126.465, -53.113, -83.952, 61.584, 66.119, -36.806]
  Call Extruder(11.08166)
  MoveL 7808 to (-40.97, 148.02, 116.27) mm, rotated rx 180 ry 0 rz 180 deg; joints [-126.491, -53.085, -84.017, 61.547, 66.121, -36.76]
  MoveL 7809 to (-40.97, 148.02, 116.27) mm, rotated rx 180 ry 0 rz 180 deg; joints [-126.491, -53.085, -84.017, 61.547, 66.121, -36.76]
  Call Extruder(11.27837)
  MoveL 7810 to (-41.02, 147.63, 116.27) mm, rotated rx 180 ry 0 rz 180 deg; joints [-126.517, -53.058, -84.082, 61.509, 66.123, -36.715]
  MoveL 7811 to (-41.02, 147.63, 116.27) mm, rotated rx 180 ry 0 rz 180 deg; joints [-126.517, -53.058, -84.082, 61.509, 66.123, -36.715]
  Call Extruder(11.47421)
  MoveL 7812 to (-41.06, 147.25, 116.27) mm, rotated rx -180 ry 0 rz 180 deg; joints [-126.543, -53.031, -84.146, 61.472, 66.126, -36.669]
  MoveL 7813 to (-41.06, 147.25, 116.27) mm, rotated rx -180 ry 0 rz 180 deg; joints [-126.543, -53.031, -84.146, 61.472, 66.126, -36.669]
  Call Extruder(11.76961)
  MoveL 7814 to (-41.11, 146.66, 116.27) mm, rotated rx 180 ry 0 rz -180 deg; joints [-126.585, -52.991, -84.242, 61.413, 66.127, -36.601]
  MoveL 7815 to (-41.11, 146.66, 116.27) mm, rotated rx 180 ry 0 rz -180 deg; joints [-126.585, -52.991, -84.242, 61.413, 66.127, -36.601]
  Call Extruder(12.06367)
  MoveL 7816 to (-41.16, 146.07, 116.27) mm, rotated rx 180 ry 0 rz -180 deg; joints [-126.628, -52.952, -84.337, 61.354, 66.129, -36.533]
  MoveL 7817 to (-41.16, 146.07, 116.27) mm, rotated rx 180 ry 0 rz -180 deg; joints [-126.628, -52.952, -84.337, 61.354, 66.129, -36.533]
  Call Extruder(12.35641)
  MoveL 7818 to (-41.2, 145.48, 116.27) mm, rotated rx -180 ry 0 rz 180 deg; joints [-126.67, -52.912, -84.433, 61.295, 66.13, -36.464]
  MoveL 7819 to (-41.2, 145.48, 116.27) mm, rotated rx -180 ry 0 rz 180 deg; joints [-126.67, -52.912, -84.433, 61.295, 66.13, -36.464]
  Call Extruder(12.92986)
  MoveL 7820 to (-41.25, 144.32, 116.27) mm, rotated rx 180 ry 0 rz 180 deg; joints [-126.759, -52.836, -84.615, 61.176, 66.128, -36.33]
  MoveL 7821 to (-41.25, 144.32, 116.27) mm, rotated rx 180 ry 0 rz 180 deg; joints [-126.759, -52.836, -84.615, 61.176, 66.128, -36.33]
  Call Extruder(13.64382)
  MoveL 7822 to (-41.29, 142.86, 116.27) mm, rotated rx 180 ry 0 rz -180 deg; joints [-126.873, -52.742, -84.841, 61.024, 66.125, -36.164]
  Call Extruder(55.70865)
  MoveL 7823 to (-41.29, 57.14, 116.27) mm, rotated rx 180 ry 0 rz 180 deg; joints [-135.148, -48.1, -96.579, 50.643, 65.803, -26.554]
  Call Extruder(56.13720)
  MoveL 7824 to (-41.27, 56.26, 116.27) mm, rotated rx -180 ry 0 rz -180 deg; joints [-135.25, -48.061, -96.683, 50.521, 65.799, -26.457]
  MoveL 7825 to (-41.27, 56.26, 116.27) mm, rotated rx -180 ry 0 rz -180 deg; joints [-135.25, -48.061, -96.683, 50.521, 65.799, -26.457]
  Call Extruder(56.71065)
  MoveL 7826 to (-41.22, 55.1, 116.27) mm, rotated rx 180 ry 0 rz 180 deg; joints [-135.387, -48.011, -96.819, 50.356, 65.793, -26.33]
  MoveL 7827 to (-41.22, 55.1, 116.27) mm, rotated rx 180 ry 0 rz 180 deg; joints [-135.387, -48.011, -96.819, 50.356, 65.793, -26.33]
  Call Extruder(57.14497)
  MoveL 7828 to (-41.18, 54.23, 116.27) mm, rotated rx 180 ry 0 rz 180 deg; joints [-135.493, -47.974, -96.92, 50.23, 65.786, -26.234]
  MoveL 7829 to (-41.18, 54.23, 116.27) mm, rotated rx 180 ry 0 rz 180 deg; joints [-135.493, -47.974, -96.92, 50.23, 65.786, -26.234]
  Call Extruder(57.43904)
  MoveL 7830 to (-41.13, 53.64, 116.27) mm, rotated rx 180 ry 0 rz 180 deg; joints [-135.566, -47.95, -96.985, 50.143, 65.78, -26.169]
  MoveL 7831 to (-41.13, 53.64, 116.27) mm, rotated rx 180 ry 0 rz 180 deg; joints [-135.566, -47.95, -96.985, 50.143, 65.78, -26.169]
  Call Extruder(57.73444)
  MoveL 7832 to (-41.09, 53.05, 116.27) mm, rotated rx 180 ry 0 rz -180 deg; joints [-135.64, -47.925, -97.051, 50.057, 65.775, -26.105]
  MoveL 7833 to (-41.09, 53.05, 116.27) mm, rotated rx 180 ry 0 rz -180 deg; joints [-135.64, -47.925, -97.051, 50.057, 65.775, -26.105]
  Call Extruder(57.98067)
  MoveL 7834 to (-41.04, 52.56, 116.27) mm, rotated rx 180 ry 0 rz 180 deg; joints [-135.701, -47.906, -97.104, 49.985, 65.769, -26.052]
  MoveL 7835 to (-41.04, 52.56, 116.27) mm, rotated rx 180 ry 0 rz 180 deg; joints [-135.701, -47.906, -97.104, 49.985, 65.769, -26.052]
  Call Extruder(58.17738)
  MoveL 7836 to (-40.99, 52.17, 116.27) mm, rotated rx 180 ry 0 rz 180 deg; joints [-135.751, -47.891, -97.145, 49.927, 65.764, -26.01]
  MoveL 7837 to (-40.99, 52.17, 116.27) mm, rotated rx 180 ry 0 rz 180 deg; joints [-135.751, -47.891, -97.145, 49.927, 65.764, -26.01]
  Call Extruder(58.37495)
  MoveL 7838 to (-40.95, 51.78, 116.27) mm, rotated rx -180 ry 0 rz -180 deg; joints [-135.801, -47.876, -97.186, 49.868, 65.758, -25.968]
  MoveL 7839 to (-40.95, 51.78, 116.27) mm, rotated rx -180 ry 0 rz -180 deg; joints [-135.801, -47.876, -97.186, 49.868, 65.758, -25.968]
  Call Extruder(58.57339)
  MoveL 7840 to (-40.9, 51.4, 116.27) mm, rotated rx 180 ry 0 rz -180 deg; joints [-135.852, -47.86, -97.227, 49.81, 65.753, -25.926]
  MoveL 7841 to (-40.9, 51.4, 116.27) mm, rotated rx 180 ry 0 rz -180 deg; joints [-135.852, -47.86, -97.227, 49.81, 65.753, -25.926]
  Call Extruder(58.77270)
  MoveL 7842 to (-40.86, 51.01, 116.27) mm, rotated rx 180 ry 0 rz 180 deg; joints [-135.902, -47.845, -97.267, 49.751, 65.748, -25.884]
  MoveL 7843 to (-40.86, 51.01, 116.27) mm, rotated rx 180 ry 0 rz 180 deg; joints [-135.902, -47.845, -97.267, 49.751, 65.748, -25.884]
  Call Extruder(58.93152)
  MoveL 7844 to (-40.81, 50.7, 116.27) mm, rotated rx 180 ry 0 rz -180 deg; joints [-135.943, -47.834, -97.298, 49.704, 65.742, -25.851]
  MoveL 7845 to (-40.81, 50.7, 116.27) mm, rotated rx 180 ry 0 rz -180 deg; joints [-135.943, -47.834, -97.298, 49.704, 65.742, -25.851]
  Call Extruder(59.09106)
  MoveL 7846 to (-40.76, 50.4, 116.27) mm, rotated rx 180 ry 0 rz -180 deg; joints [-135.984, -47.823, -97.329, 49.657, 65.737, -25.818]
  MoveL 7847 to (-40.76, 50.4, 116.27) mm, rotated rx 180 ry 0 rz -180 deg; joints [-135.984, -47.823, -97.329, 49.657, 65.737, -25.818]
  Call Extruder(59.25133)
  MoveL 7848 to (-40.71, 50.09, 116.27) mm, rotated rx 180 ry 0 rz 180 deg; joints [-136.025, -47.812, -97.359, 49.61, 65.731, -25.786]
  MoveL 7849 to (-40.71, 50.09, 116.27) mm, rotated rx 180 ry 0 rz 180 deg; joints [-136.025, -47.812, -97.359, 49.61, 65.731, -25.786]
  Call Extruder(59.41232)
  MoveL 7850 to (-40.66, 49.79, 116.27) mm, rotated rx 180 ry 0 rz -180 deg; joints [-136.067, -47.8, -97.39, 49.562, 65.726, -25.753]
  MoveL 7851 to (-40.66, 49.79, 116.27) mm, rotated rx 180 ry 0 rz -180 deg; joints [-136.067, -47.8, -97.39, 49.562, 65.726, -25.753]
  Call Extruder(59.57405)
  MoveL 7852 to (-40.61, 49.48, 116.27) mm, rotated rx 180 ry 0 rz -180 deg; joints [-136.108, -47.789, -97.42, 49.515, 65.721, -25.72]
  MoveL 7853 to (-40.61, 49.48, 116.27) mm, rotated rx 180 ry 0 rz -180 deg; joints [-136.108, -47.789, -97.42, 49.515, 65.721, -25.72]
  Call Extruder(59.73650)
  MoveL 7854 to (-40.57, 49.17, 116.27) mm, rotated rx -180 ry 0 rz -180 deg; joints [-136.149, -47.778, -97.45, 49.468, 65.715, -25.687]
  MoveL 7855 to (-40.57, 49.17, 116.27) mm, rotated rx -180 ry 0 rz -180 deg; joints [-136.149, -47.778, -97.45, 49.468, 65.715, -25.687]
  Call Extruder(59.87043)
  MoveL 7856 to (-40.52, 48.93, 116.27) mm, rotated rx 180 ry 0 rz -180 deg; joints [-136.184, -47.769, -97.474, 49.428, 65.71, -25.66]
  MoveL 7857 to (-40.52, 48.93, 116.27) mm, rotated rx 180 ry 0 rz -180 deg; joints [-136.184, -47.769, -97.474, 49.428, 65.71, -25.66]
  Call Extruder(60.00496)
  MoveL 7858 to (-40.47, 48.68, 116.27) mm, rotated rx 180 ry 0 rz 180 deg; joints [-136.219, -47.761, -97.498, 49.388, 65.704, -25.634]
  MoveL 7859 to (-40.47, 48.68, 116.27) mm, rotated rx 180 ry 0 rz 180 deg; joints [-136.219, -47.761, -97.498, 49.388, 65.704, -25.634]
  Call Extruder(60.14011)
  MoveL 7860 to (-40.42, 48.43, 116.27) mm, rotated rx -180 ry 0 rz 180 deg; joints [-136.254, -47.752, -97.521, 49.349, 65.699, -25.607]
  MoveL 7861 to (-40.42, 48.43, 116.27) mm, rotated rx -180 ry 0 rz 180 deg; joints [-136.254, -47.752, -97.521, 49.349, 65.699, -25.607]
  Call Extruder(60.27586)
  MoveL 7862 to (-40.37, 48.18, 116.27) mm, rotated rx 180 ry 0 rz 180 deg; joints [-136.288, -47.743, -97.545, 49.309, 65.694, -25.581]
  MoveL 7863 to (-40.37, 48.18, 116.27) mm, rotated rx 180 ry 0 rz 180 deg; joints [-136.288, -47.743, -97.545, 49.309, 65.694, -25.581]
  Call Extruder(60.41223)
  MoveL 7864 to (-40.32, 47.93, 116.27) mm, rotated rx -180 ry 0 rz -180 deg; joints [-136.323, -47.735, -97.568, 49.27, 65.688, -25.554]
  MoveL 7865 to (-40.32, 47.93, 116.27) mm, rotated rx -180 ry 0 rz -180 deg; joints [-136.323, -47.735, -97.568, 49.27, 65.688, -25.554]
  Call Extruder(60.54920)
  MoveL 7866 to (-40.27, 47.68, 116.27) mm, rotated rx 180 ry 0 rz -180 deg; joints [-136.358, -47.726, -97.591, 49.23, 65.683, -25.528]
  MoveL 7867 to (-40.27, 47.68, 116.27) mm, rotated rx 180 ry 0 rz -180 deg; joints [-136.358, -47.726, -97.591, 49.23, 65.683, -25.528]
  Call Extruder(60.68679)
  MoveL 7868 to (-40.22, 47.43, 116.27) mm, rotated rx 180 ry 0 rz 180 deg; joints [-136.393, -47.718, -97.615, 49.19, 65.677, -25.501]
  MoveL 7869 to (-40.22, 47.43, 116.27) mm, rotated rx 180 ry 0 rz 180 deg; joints [-136.393, -47.718, -97.615, 49.19, 65.677, -25.501]
  Call Extruder(60.80052)
  MoveL 7870 to (-40.17, 47.23, 116.27) mm, rotated rx 180 ry 0 rz -180 deg; joints [-136.422, -47.711, -97.633, 49.158, 65.673, -25.479]
  MoveL 7871 to (-40.17, 47.23, 116.27) mm, rotated rx 180 ry 0 rz -180 deg; joints [-136.422, -47.711, -97.633, 49.158, 65.673, -25.479]
  Call Extruder(60.91470)
  MoveL 7872 to (-40.13, 47.02, 116.27) mm, rotated rx 180 ry 0 rz 180 deg; joints [-136.452, -47.704, -97.652, 49.124, 65.668, -25.458]
  MoveL 7873 to (-40.13, 47.02, 116.27) mm, rotated rx 180 ry 0 rz 180 deg; joints [-136.452, -47.704, -97.652, 49.124, 65.668, -25.458]
  Call Extruder(61.02933)
  MoveL 7874 to (-40.08, 46.82, 116.27) mm, rotated rx 180 ry 0 rz -180 deg; joints [-136.481, -47.697, -97.671, 49.092, 65.663, -25.436]
  MoveL 7875 to (-40.08, 46.82, 116.27) mm, rotated rx 180 ry 0 rz -180 deg; joints [-136.481, -47.697, -97.671, 49.092, 65.663, -25.436]
  Call Extruder(61.14442)
  MoveL 7876 to (-40.04, 46.61, 116.27) mm, rotated rx -180 ry 0 rz 180 deg; joints [-136.51, -47.69, -97.689, 49.059, 65.658, -25.414]
  MoveL 7877 to (-40.04, 46.61, 116.27) mm, rotated rx -180 ry 0 rz 180 deg; joints [-136.51, -47.69, -97.689, 49.059, 65.658, -25.414]
  Call Extruder(61.26666)
  MoveL 7878 to (-39.98, 46.4, 116.27) mm, rotated rx -180 ry 0 rz 180 deg; joints [-136.542, -47.684, -97.707, 49.023, 65.652, -25.392]
  MoveL 7879 to (-39.98, 46.4, 116.27) mm, rotated rx -180 ry 0 rz 180 deg; joints [-136.542, -47.684, -97.707, 49.023, 65.652, -25.392]
  Call Extruder(61.39632)
  MoveL 7880 to (-39.92, 46.18, 116.27) mm, rotated rx -180 ry 0 rz 180 deg; joints [-136.576, -47.677, -97.725, 48.985, 65.645, -25.368]
  MoveL 7881 to (-39.92, 46.18, 116.27) mm, rotated rx -180 ry 0 rz 180 deg; joints [-136.576, -47.677, -97.725, 48.985, 65.645, -25.368]
  Call Extruder(61.52655)
  MoveL 7882 to (-39.85, 45.95, 116.27) mm, rotated rx 180 ry 0 rz -180 deg; joints [-136.61, -47.671, -97.743, 48.948, 65.638, -25.345]
  MoveL 7883 to (-39.85, 45.95, 116.27) mm, rotated rx 180 ry 0 rz -180 deg; joints [-136.61, -47.671, -97.743, 48.948, 65.638, -25.345]
  Call Extruder(61.65735)
  MoveL 7884 to (-39.78, 45.73, 116.27) mm, rotated rx -180 ry 0 rz 180 deg; joints [-136.644, -47.664, -97.761, 48.91, 65.631, -25.322]
  MoveL 7885 to (-39.78, 45.73, 116.27) mm, rotated rx -180 ry 0 rz 180 deg; joints [-136.644, -47.664, -97.761, 48.91, 65.631, -25.322]
  Call Extruder(61.78871)
  MoveL 7886 to (-39.71, 45.5, 116.27) mm, rotated rx -180 ry 0 rz 180 deg; joints [-136.678, -47.657, -97.779, 48.872, 65.624, -25.298]
  MoveL 7887 to (-39.71, 45.5, 116.27) mm, rotated rx -180 ry 0 rz 180 deg; joints [-136.678, -47.657, -97.779, 48.872, 65.624, -25.298]
  Call Extruder(61.90061)
  MoveL 7888 to (-39.65, 45.32, 116.27) mm, rotated rx 180 ry 0 rz -180 deg; joints [-136.707, -47.652, -97.794, 48.84, 65.617, -25.279]
  MoveL 7889 to (-39.65, 45.32, 116.27) mm, rotated rx 180 ry 0 rz -180 deg; joints [-136.707, -47.652, -97.794, 48.84, 65.617, -25.279]
  Call Extruder(62.01295)
  MoveL 7890 to (-39.59, 45.13, 116.27) mm, rotated rx 180 ry 0 rz 180 deg; joints [-136.737, -47.647, -97.808, 48.808, 65.611, -25.259]
  MoveL 7891 to (-39.59, 45.13, 116.27) mm, rotated rx 180 ry 0 rz 180 deg; joints [-136.737, -47.647, -97.808, 48.808, 65.611, -25.259]
  Call Extruder(62.12574)
  MoveL 7892 to (-39.53, 44.94, 116.27) mm, rotated rx 180 ry 0 rz 180 deg; joints [-136.766, -47.642, -97.823, 48.775, 65.604, -25.239]
  MoveL 7893 to (-39.53, 44.94, 116.27) mm, rotated rx 180 ry 0 rz 180 deg; joints [-136.766, -47.642, -97.823, 48.775, 65.604, -25.239]
  Call Extruder(62.23898)
  MoveL 7894 to (-39.47, 44.75, 116.27) mm, rotated rx 180 ry 0 rz -180 deg; joints [-136.796, -47.636, -97.837, 48.743, 65.598, -25.22]
  MoveL 7895 to (-39.47, 44.75, 116.27) mm, rotated rx 180 ry 0 rz -180 deg; joints [-136.796, -47.636, -97.837, 48.743, 65.598, -25.22]
  Call Extruder(62.35266)
  MoveL 7896 to (-39.41, 44.56, 116.27) mm, rotated rx 180 ry 0 rz 180 deg; joints [-136.825, -47.631, -97.852, 48.711, 65.591, -25.2]
  MoveL 7897 to (-39.41, 44.56, 116.27) mm, rotated rx 180 ry 0 rz 180 deg; joints [-136.825, -47.631, -97.852, 48.711, 65.591, -25.2]
  Call Extruder(62.53462)
  MoveL 7898 to (-39.29, 44.27, 116.27) mm, rotated rx 180 ry 0 rz -180 deg; joints [-136.873, -47.624, -97.871, 48.659, 65.579, -25.17]
  MoveL 7899 to (-39.29, 44.27, 116.27) mm, rotated rx 180 ry 0 rz -180 deg; joints [-136.873, -47.624, -97.871, 48.659, 65.579, -25.17]
  Call Extruder(62.71734)
  MoveL 7900 to (-39.17, 43.98, 116.27) mm, rotated rx -180 ry 0 rz 180 deg; joints [-136.922, -47.617, -97.89, 48.606, 65.566, -25.14]
  MoveL 7901 to (-39.17, 43.98, 116.27) mm, rotated rx -180 ry 0 rz 180 deg; joints [-136.922, -47.617, -97.89, 48.606, 65.566, -25.14]
  Call Extruder(62.88775)
  MoveL 7902 to (-39.05, 43.71, 116.27) mm, rotated rx -180 ry 0 rz 180 deg; joints [-136.967, -47.611, -97.907, 48.558, 65.554, -25.113]
  MoveL 7903 to (-39.05, 43.71, 116.27) mm, rotated rx -180 ry 0 rz 180 deg; joints [-136.967, -47.611, -97.907, 48.558, 65.554, -25.113]
  Call Extruder(63.04573)
  MoveL 7904 to (-38.94, 43.46, 116.27) mm, rotated rx 180 ry 0 rz 180 deg; joints [-137.009, -47.605, -97.923, 48.513, 65.543, -25.087]
  MoveL 7905 to (-38.94, 43.46, 116.27) mm, rotated rx 180 ry 0 rz 180 deg; joints [-137.009, -47.605, -97.923, 48.513, 65.543, -25.087]
  Call Extruder(63.20432)
  MoveL 7906 to (-38.84, 43.21, 116.27) mm, rotated rx 180 ry 0 rz 180 deg; joints [-137.05, -47.599, -97.939, 48.468, 65.532, -25.062]
  MoveL 7907 to (-38.84, 43.21, 116.27) mm, rotated rx 180 ry 0 rz 180 deg; joints [-137.05, -47.599, -97.939, 48.468, 65.532, -25.062]
  Call Extruder(63.41049)
  MoveL 7908 to (-38.66, 42.91, 116.27) mm, rotated rx 180 ry 0 rz -180 deg; joints [-137.107, -47.594, -97.952, 48.409, 65.514, -25.031]
  MoveL 7909 to (-38.66, 42.91, 116.27) mm, rotated rx 180 ry 0 rz -180 deg; joints [-137.107, -47.594, -97.952, 48.409, 65.514, -25.031]
  Call Extruder(63.61743)
  MoveL 7910 to (-38.49, 42.6, 116.27) mm, rotated rx 180 ry 0 rz -180 deg; joints [-137.163, -47.589, -97.966, 48.35, 65.496, -25.001]
  MoveL 7911 to (-38.49, 42.6, 116.27) mm, rotated rx 180 ry 0 rz -180 deg; joints [-137.163, -47.589, -97.966, 48.35, 65.496, -25.001]
  Call Extruder(63.82516)
  MoveL 7912 to (-38.31, 42.3, 116.27) mm, rotated rx 180 ry 0 rz 180 deg; joints [-137.219, -47.584, -97.979, 48.291, 65.478, -24.971]
  MoveL 7913 to (-38.31, 42.3, 116.27) mm, rotated rx 180 ry 0 rz 180 deg; joints [-137.219, -47.584, -97.979, 48.291, 65.478, -24.971]
  Call Extruder(64.03366)
  MoveL 7914 to (-38.13, 41.99, 116.27) mm, rotated rx 180 ry 0 rz 180 deg; joints [-137.275, -47.58, -97.992, 48.232, 65.46, -24.941]
  MoveL 7915 to (-38.13, 41.99, 116.27) mm, rotated rx 180 ry 0 rz 180 deg; joints [-137.275, -47.58, -97.992, 48.232, 65.46, -24.941]
  Call Extruder(64.21320)
  MoveL 7916 to (-37.96, 41.75, 116.27) mm, rotated rx 180 ry 0 rz 180 deg; joints [-137.324, -47.577, -97.999, 48.182, 65.442, -24.917]
  MoveL 7917 to (-37.96, 41.75, 116.27) mm, rotated rx 180 ry 0 rz 180 deg; joints [-137.324, -47.577, -97.999, 48.182, 65.442, -24.917]
  Call Extruder(64.54664)
  MoveL 7918 to (-37.63, 41.3, 116.27) mm, rotated rx 180 ry 0 rz 180 deg; joints [-137.415, -47.573, -98.009, 48.089, 65.408, -24.874]
  MoveL 7919 to (-37.63, 41.3, 116.27) mm, rotated rx 180 ry 0 rz 180 deg; joints [-137.415, -47.573, -98.009, 48.089, 65.408, -24.874]
  Call Extruder(64.88126)
  MoveL 7920 to (-37.3, 40.85, 116.27) mm, rotated rx 180 ry 0 rz 180 deg; joints [-137.506, -47.569, -98.02, 47.996, 65.374, -24.83]
  Call Extruder(65.70919)
  MoveL 7921 to (-36.39, 39.81, 116.27) mm, rotated rx 180 ry 0 rz -180 deg; joints [-137.733, -47.568, -98.025, 47.768, 65.281, -24.734]
  Call Extruder(66.53710)
  MoveL 7922 to (-35.35, 38.9, 116.27) mm, rotated rx -180 ry 0 rz -180 deg; joints [-137.958, -47.578, -97.998, 47.549, 65.176, -24.653]
  Call Extruder(66.70441)
  MoveL 7923 to (-35.13, 38.73, 116.27) mm, rotated rx 180 ry 0 rz 180 deg; joints [-138.003, -47.581, -97.988, 47.506, 65.153, -24.639]
  MoveL 7924 to (-35.13, 38.73, 116.27) mm, rotated rx 180 ry 0 rz 180 deg; joints [-138.003, -47.581, -97.988, 47.506, 65.153, -24.639]
  Call Extruder(67.03783)
  MoveL 7925 to (-34.68, 38.4, 116.27) mm, rotated rx -180 ry 0 rz -180 deg; joints [-138.092, -47.588, -97.968, 47.421, 65.107, -24.612]
  MoveL 7926 to (-34.68, 38.4, 116.27) mm, rotated rx -180 ry 0 rz -180 deg; joints [-138.092, -47.588, -97.968, 47.421, 65.107, -24.612]
  Call Extruder(67.37007)
  MoveL 7927 to (-34.23, 38.08, 116.27) mm, rotated rx 180 ry 0 rz -180 deg; joints [-138.182, -47.596, -97.948, 47.335, 65.061, -24.584]
  MoveL 7928 to (-34.23, 38.08, 116.27) mm, rotated rx 180 ry 0 rz -180 deg; joints [-138.182, -47.596, -97.948, 47.335, 65.061, -24.584]
  Call Extruder(67.48778)
  MoveL 7929 to (-34.05, 37.98, 116.27) mm, rotated rx -180 ry 0 rz 180 deg; joints [-138.213, -47.6, -97.937, 47.307, 65.044, -24.577]
  MoveL 7930 to (-34.05, 37.98, 116.27) mm, rotated rx -180 ry 0 rz 180 deg; joints [-138.213, -47.6, -97.937, 47.307, 65.044, -24.577]
  Call Extruder(67.69550)
  MoveL 7931 to (-33.75, 37.8, 116.27) mm, rotated rx 180 ry 0 rz 180 deg; joints [-138.267, -47.606, -97.919, 47.256, 65.013, -24.563]
  MoveL 7932 to (-33.75, 37.8, 116.27) mm, rotated rx 180 ry 0 rz 180 deg; joints [-138.267, -47.606, -97.919, 47.256, 65.013, -24.563]
  Call Extruder(67.90244)
  MoveL 7933 to (-33.45, 37.63, 116.27) mm, rotated rx -180 ry 0 rz 180 deg; joints [-138.322, -47.613, -97.9, 47.205, 64.982, -24.55]
  MoveL 7934 to (-33.45, 37.63, 116.27) mm, rotated rx -180 ry 0 rz 180 deg; joints [-138.322, -47.613, -97.9, 47.205, 64.982, -24.55]
  Call Extruder(68.10860)
  MoveL 7935 to (-33.14, 37.45, 116.27) mm, rotated rx -180 ry 0 rz 180 deg; joints [-138.376, -47.62, -97.881, 47.155, 64.951, -24.537]
  MoveL 7936 to (-33.14, 37.45, 116.27) mm, rotated rx -180 ry 0 rz 180 deg; joints [-138.376, -47.62, -97.881, 47.155, 64.951, -24.537]
  Call Extruder(68.29029)
  MoveL 7937 to (-32.86, 37.31, 116.27) mm, rotated rx 180 ry 0 rz 180 deg; joints [-138.424, -47.627, -97.861, 47.111, 64.923, -24.526]
  MoveL 7938 to (-32.86, 37.31, 116.27) mm, rotated rx 180 ry 0 rz 180 deg; joints [-138.424, -47.627, -97.861, 47.111, 64.923, -24.526]
  Call Extruder(68.44829)
  MoveL 7939 to (-32.62, 37.2, 116.27) mm, rotated rx 180 ry 0 rz -180 deg; joints [-138.464, -47.635, -97.842, 47.075, 64.898, -24.519]
  MoveL 7940 to (-32.62, 37.2, 116.27) mm, rotated rx 180 ry 0 rz -180 deg; joints [-138.464, -47.635, -97.842, 47.075, 64.898, -24.519]
  Call Extruder(68.60569)
  MoveL 7941 to (-32.37, 37.1, 116.27) mm, rotated rx 180 ry 0 rz 180 deg; joints [-138.504, -47.642, -97.822, 47.039, 64.873, -24.512]
  MoveL 7942 to (-32.37, 37.1, 116.27) mm, rotated rx 180 ry 0 rz 180 deg; joints [-138.504, -47.642, -97.822, 47.039, 64.873, -24.512]
  Call Extruder(68.78840)
  MoveL 7943 to (-32.07, 36.98, 116.27) mm, rotated rx 180 ry 0 rz 180 deg; joints [-138.551, -47.651, -97.798, 46.998, 64.843, -24.505]
  MoveL 7944 to (-32.07, 36.98, 116.27) mm, rotated rx 180 ry 0 rz 180 deg; joints [-138.551, -47.651, -97.798, 46.998, 64.843, -24.505]
  Call Extruder(68.97035)
  MoveL 7945 to (-31.78, 36.85, 116.27) mm, rotated rx 180 ry 0 rz 180 deg; joints [-138.597, -47.659, -97.774, 46.956, 64.813, -24.497]
  MoveL 7946 to (-31.78, 36.85, 116.27) mm, rotated rx 180 ry 0 rz 180 deg; joints [-138.597, -47.659, -97.774, 46.956, 64.813, -24.497]
  Call Extruder(69.11768)
  MoveL 7947 to (-31.54, 36.76, 116.27) mm, rotated rx 180 ry 0 rz 180 deg; joints [-138.634, -47.667, -97.753, 46.923, 64.789, -24.492]
  MoveL 7948 to (-31.54, 36.76, 116.27) mm, rotated rx 180 ry 0 rz 180 deg; joints [-138.634, -47.667, -97.753, 46.923, 64.789, -24.492]
  Call Extruder(69.23091)
  MoveL 7949 to (-31.35, 36.7, 116.27) mm, rotated rx -180 ry 0 rz 180 deg; joints [-138.662, -47.673, -97.736, 46.899, 64.77, -24.489]
  MoveL 7950 to (-31.35, 36.7, 116.27) mm, rotated rx -180 ry 0 rz 180 deg; joints [-138.662, -47.673, -97.736, 46.899, 64.77, -24.489]
  Call Extruder(69.34371)
  MoveL 7951 to (-31.17, 36.64, 116.27) mm, rotated rx 180 ry 0 rz -180 deg; joints [-138.69, -47.68, -97.719, 46.875, 64.751, -24.486]
  MoveL 7952 to (-31.17, 36.64, 116.27) mm, rotated rx 180 ry 0 rz -180 deg; joints [-138.69, -47.68, -97.719, 46.875, 64.751, -24.486]
  Call Extruder(69.45605)
  MoveL 7953 to (-30.98, 36.58, 116.27) mm, rotated rx 180 ry 0 rz -180 deg; joints [-138.718, -47.686, -97.701, 46.851, 64.732, -24.483]
  MoveL 7954 to (-30.98, 36.58, 116.27) mm, rotated rx 180 ry 0 rz -180 deg; joints [-138.718, -47.686, -97.701, 46.851, 64.732, -24.483]
  Call Extruder(69.56796)
  MoveL 7955 to (-30.79, 36.52, 116.27) mm, rotated rx 180 ry 0 rz -180 deg; joints [-138.745, -47.692, -97.684, 46.827, 64.713, -24.48]
  MoveL 7956 to (-30.79, 36.52, 116.27) mm, rotated rx 180 ry 0 rz -180 deg; joints [-138.745, -47.692, -97.684, 46.827, 64.713, -24.48]
  Call Extruder(69.68936)
  MoveL 7957 to (-30.58, 36.45, 116.27) mm, rotated rx 180 ry 0 rz 180 deg; joints [-138.776, -47.699, -97.665, 46.8, 64.692, -24.476]
  MoveL 7958 to (-30.58, 36.45, 116.27) mm, rotated rx 180 ry 0 rz 180 deg; joints [-138.776, -47.699, -97.665, 46.8, 64.692, -24.476]
  Call Extruder(69.82015)
  MoveL 7959 to (-30.36, 36.39, 116.27) mm, rotated rx -180 ry 0 rz 180 deg; joints [-138.808, -47.707, -97.643, 46.772, 64.669, -24.473]
  MoveL 7960 to (-30.36, 36.39, 116.27) mm, rotated rx -180 ry 0 rz 180 deg; joints [-138.808, -47.707, -97.643, 46.772, 64.669, -24.473]
  Call Extruder(69.95037)
  MoveL 7961 to (-30.14, 36.32, 116.27) mm, rotated rx 180 ry 0 rz 180 deg; joints [-138.84, -47.715, -97.622, 46.745, 64.647, -24.47]
  MoveL 7962 to (-30.14, 36.32, 116.27) mm, rotated rx 180 ry 0 rz 180 deg; joints [-138.84, -47.715, -97.622, 46.745, 64.647, -24.47]
  Call Extruder(70.08003)
  MoveL 7963 to (-29.91, 36.25, 116.27) mm, rotated rx 180 ry 0 rz -180 deg; joints [-138.873, -47.723, -97.601, 46.717, 64.624, -24.467]
  MoveL 7964 to (-29.91, 36.25, 116.27) mm, rotated rx 180 ry 0 rz -180 deg; joints [-138.873, -47.723, -97.601, 46.717, 64.624, -24.467]
  Call Extruder(70.20913)
  MoveL 7965 to (-29.69, 36.18, 116.27) mm, rotated rx -180 ry 0 rz -180 deg; joints [-138.905, -47.731, -97.579, 46.689, 64.602, -24.464]
  MoveL 7966 to (-29.69, 36.18, 116.27) mm, rotated rx -180 ry 0 rz -180 deg; joints [-138.905, -47.731, -97.579, 46.689, 64.602, -24.464]
  Call Extruder(70.32420)
  MoveL 7967 to (-29.48, 36.14, 116.27) mm, rotated rx 180 ry 0 rz 180 deg; joints [-138.932, -47.738, -97.558, 46.666, 64.581, -24.463]
  MoveL 7968 to (-29.48, 36.14, 116.27) mm, rotated rx 180 ry 0 rz 180 deg; joints [-138.932, -47.738, -97.558, 46.666, 64.581, -24.463]
  Call Extruder(70.43882)
  MoveL 7969 to (-29.28, 36.09, 116.27) mm, rotated rx -180 ry 0 rz 180 deg; joints [-138.96, -47.746, -97.537, 46.643, 64.56, -24.462]
  MoveL 7970 to (-29.28, 36.09, 116.27) mm, rotated rx -180 ry 0 rz 180 deg; joints [-138.96, -47.746, -97.537, 46.643, 64.56, -24.462]
  Call Extruder(70.55299)
  MoveL 7971 to (-29.08, 36.05, 116.27) mm, rotated rx -180 ry 0 rz -180 deg; joints [-138.987, -47.754, -97.515, 46.62, 64.54, -24.462]
  MoveL 7972 to (-29.08, 36.05, 116.27) mm, rotated rx -180 ry 0 rz -180 deg; joints [-138.987, -47.754, -97.515, 46.62, 64.54, -24.462]
  Call Extruder(70.66671)
  MoveL 7973 to (-28.87, 36, 116.27) mm, rotated rx 180 ry 0 rz -180 deg; joints [-139.014, -47.762, -97.494, 46.597, 64.519, -24.461]
  MoveL 7974 to (-28.87, 36, 116.27) mm, rotated rx 180 ry 0 rz -180 deg; joints [-139.014, -47.762, -97.494, 46.597, 64.519, -24.461]
  Call Extruder(70.79213)
  MoveL 7975 to (-28.64, 35.96, 116.27) mm, rotated rx 180 ry 0 rz 180 deg; joints [-139.044, -47.771, -97.47, 46.573, 64.496, -24.46]
  MoveL 7976 to (-28.64, 35.96, 116.27) mm, rotated rx 180 ry 0 rz 180 deg; joints [-139.044, -47.771, -97.47, 46.573, 64.496, -24.46]
  Call Extruder(70.92911)
  MoveL 7977 to (-28.4, 35.91, 116.27) mm, rotated rx 180 ry 0 rz -180 deg; joints [-139.077, -47.781, -97.443, 46.546, 64.471, -24.459]
  MoveL 7978 to (-28.4, 35.91, 116.27) mm, rotated rx 180 ry 0 rz -180 deg; joints [-139.077, -47.781, -97.443, 46.546, 64.471, -24.459]
  Call Extruder(71.06547)
  MoveL 7979 to (-28.15, 35.86, 116.27) mm, rotated rx 180 ry 0 rz 180 deg; joints [-139.109, -47.791, -97.416, 46.519, 64.446, -24.459]
  MoveL 7980 to (-28.15, 35.86, 116.27) mm, rotated rx 180 ry 0 rz 180 deg; joints [-139.109, -47.791, -97.416, 46.519, 64.446, -24.459]
  Call Extruder(71.20123)
  MoveL 7981 to (-27.9, 35.81, 116.27) mm, rotated rx 180 ry 0 rz 180 deg; joints [-139.142, -47.801, -97.389, 46.491, 64.421, -24.458]
  MoveL 7982 to (-27.9, 35.81, 116.27) mm, rotated rx 180 ry 0 rz 180 deg; joints [-139.142, -47.801, -97.389, 46.491, 64.421, -24.458]
  Call Extruder(71.33638)
  MoveL 7983 to (-27.65, 35.76, 116.27) mm, rotated rx 180 ry 0 rz 180 deg; joints [-139.174, -47.81, -97.362, 46.465, 64.395, -24.458]
  MoveL 7984 to (-27.65, 35.76, 116.27) mm, rotated rx 180 ry 0 rz 180 deg; joints [-139.174, -47.81, -97.362, 46.465, 64.395, -24.458]
  Call Extruder(71.47091)
  MoveL 7985 to (-27.4, 35.71, 116.27) mm, rotated rx 180 ry 0 rz 180 deg; joints [-139.207, -47.82, -97.335, 46.438, 64.37, -24.457]
